LIN {X 0,Y 188.543,Z 754.958,A -85,B 0,C 180,E1 -22070.169,E2 -22070.169} C_VEL
LIN {X 0,Y 190.971,Z 747.164,A -85,B 0,C 180,E1 -22073.069,E2 -22073.069} C_VEL
LIN {X 0,Y 193.636,Z 737.842,A -85,B 0,C 180,E1 -22075.819,E2 -22075.819} C_VEL
LIN {X 0,Y 196.619,Z 727.143,A -85,B 0,C 180,E1 -22078.268,E2 -22078.268} C_VEL
LIN {X 0,Y 199.32,Z 716.514,A -85,B 0,C 180,E1 -22080.162,E2 -22080.162} C_VEL
LIN {X 0,Y 201.799,Z 704.647,A -85,B 0,C 180,E1 -22081.786,E2 -22081.786} C_VEL
LIN {X 0,Y 203.932,Z 692.297,A -85,B 0,C 180,E1 -22083.02,E2 -22083.02} C_VEL
LIN {X 0,Y 205.572,Z 679.263,A -85,B 0,C 180,E1 -22083.923,E2 -22083.923} C_VEL
LIN {X 0,Y 206.507,Z 665.005,A -85,B 0,C 180,E1 -22084.513,E2 -22084.513} C_VEL
LIN {X 0,Y 208.41,Z 623.369,A -85,B 0,C 180,E1 -22085.857,E2 -22085.857} C_VEL
LIN {X 0,Y 206.584,Z 608.008,A -85,B 0,C 180,E1 -22086.831,E2 -22086.831} C_VEL
LIN {X 0,Y 200.505,Z 592.715,A -85,B 0,C 180,E1 -22088.711,E2 -22088.711} C_VEL
LIN {X 0,Y 194.742,Z 580.478,A -85,B 0,C 180,E1 -22090.545,E2 -22090.545} C_VEL
LIN {X 0,Y 188.91,Z 569.734,A -85,B 0,C 180,E1 -22092.487,E2 -22092.487} C_VEL
LIN {X 0,Y 186.505,Z 565.259,A -85,B 0,C 180,E1 -22093.393,E2 -22093.393} C_VEL
LIN {X 0,Y 185.509,Z 561.374,A -85,B 0,C 180,E1 -22096.038,E2 -22096.038} C_VEL
LIN {X 0,Y 185.527,Z 561.37,A -85,B 0,C 180,E1 -22099.911,E2 -22099.911} C_VEL
LIN {X 0,Y 185.557,Z 561.366,A -85,B 0,C 180,E1 -22102.699,E2 -22102.699} C_VEL
LIN {X 0,Y 185.542,Z 561.366,A -85,B 0,C 180,E1 -22107.975,E2 -22107.975} C_VEL
LIN {X 0,Y 185.579,Z 561.365,A -85,B 0,C 180,E1 -22110.575,E2 -22110.575} C_VEL
LIN {X 0,Y 185.577,Z 561.365,A -85,B 0,C 180,E1 -22115.381,E2 -22115.381} C_VEL
LIN {X 0,Y 185.67,Z 561.351,A -85,B 0,C 180,E1 -22121.134,E2 -22121.134} C_VEL
LIN {X 0,Y 185.689,Z 561.353,A -85,B 0,C 180,E1 -22124.637,E2 -22124.637} C_VEL
LIN {X 0,Y 185.92,Z 561.313,A -85,B 0,C 180,E1 -22129.359,E2 -22129.359} C_VEL
LIN {X 0,Y 185.956,Z 561.316,A -85,B 0,C 180,E1 -22133.49,E2 -22133.49} C_VEL
LIN {X 0,Y 186.203,Z 561.289,A -85,B 0,C 180,E1 -22137.837,E2 -22137.837} C_VEL
LIN {X 0,Y 186.402,Z 561.263,A -85,B 0,C 180,E1 -22140,E2 -22140} C_VEL
LIN {X 0,Y 185.918,Z 561.321,A -85,B 0,C 180,E1 -22144.336,E2 -22144.336} C_VEL
LIN {X 0,Y 185.983,Z 561.305,A -85,B 0,C 180,E1 -22148.694,E2 -22148.694} C_VEL
LIN {X 0,Y 185.725,Z 561.339,A -85,B 0,C 180,E1 -22153.124,E2 -22153.124} C_VEL
LIN {X 0,Y 185.687,Z 561.346,A -85,B 0,C 180,E1 -22157.626,E2 -22157.626} C_VEL
LIN {X 0,Y 185.594,Z 561.358,A -85,B 0,C 180,E1 -22162.252,E2 -22162.252} C_VEL
LIN {X 0,Y 185.56,Z 561.363,A -85,B 0,C 180,E1 -22167.033,E2 -22167.033} C_VEL
LIN {X 0,Y 185.577,Z 561.369,A -85,B 0,C 180,E1 -22169.494,E2 -22169.494} C_VEL
LIN {X 0,Y 185.517,Z 561.375,A -85,B 0,C 180,E1 -22174.629,E2 -22174.629} C_VEL
LIN {X 0,Y 185.542,Z 561.349,A -85,B 0,C 180,E1 -22177.305,E2 -22177.305} C_VEL
LIN {X 0,Y 185.502,Z 561.377,A -85,B 0,C 180,E1 -22180.737,E2 -22180.737} C_VEL
LIN {X 0,Y 185.557,Z 561.366,A -85,B 0,C 180,E1 -22186.024,E2 -22186.024} C_VEL
LIN {X 0,Y 185.54,Z 561.371,A -85,B 0,C 180,E1 -22190.642,E2 -22190.642} C_VEL
LIN {X 0,Y 186.562,Z 564.249,A -85,B 0,C 180,E1 -22191.08,E2 -22191.08} C_VEL
LIN {X 0,Y 188.397,Z 566.543,A -85,B 0,C 180,E1 -22191.68,E2 -22191.68} C_VEL
LIN {X 0,Y 190.496,Z 569.807,A -85,B 0,C 180,E1 -22192.378,E2 -22192.378} C_VEL
LIN {X 0,Y 198.121,Z 582.425,A -85,B 0,C 180,E1 -22194.771,E2 -22194.771} C_VEL
LIN {X 0,Y 202.401,Z 590.493,A -85,B 0,C 180,E1 -22196.048,E2 -22196.048} C_VEL
LIN {X 0,Y 208.127,Z 604.639,A -85,B 0,C 180,E1 -22197.782,E2 -22197.782} C_VEL
LIN {X 0,Y 209.093,Z 607.323,A -85,B 0,C 180,E1 -22198.074,E2 -22198.074} C_VEL
LIN {X 0,Y 206.377,Z 664.41,A -85,B 0,C 180,E1 -22199.96,E2 -22199.96} C_VEL
LIN {X 0,Y 205.136,Z 677.197,A -85,B 0,C 180,E1 -22200.724,E2 -22200.724} C_VEL
LIN {X 0,Y 203.324,Z 690.286,A -85,B 0,C 180,E1 -22201.905,E2 -22201.905} C_VEL
LIN {X 0,Y 201.181,Z 701.437,A -85,B 0,C 180,E1 -22203.272,E2 -22203.272} C_VEL
LIN {X 0,Y 198.677,Z 712.971,A -85,B 0,C 180,E1 -22205.162,E2 -22205.162} C_VEL
LIN {X 0,Y 195.999,Z 723.355,A -85,B 0,C 180,E1 -22207.328,E2 -22207.328} C_VEL
LIN {X 0,Y 193.122,Z 732.726,A -85,B 0,C 180,E1 -22209.775,E2 -22209.775} C_VEL
LIN {X 0,Y 190.815,Z 740.39,A -85,B 0,C 180,E1 -22212.311,E2 -22212.311} C_VEL
LIN {X 0,Y 188.536,Z 747.886,A -85,B 0,C 180,E1 -22215.427,E2 -22215.427} C_VEL
LIN {X 0,Y 186.376,Z 754.818,A -85,B 0,C 180,E1 -22219.132,E2 -22219.132} C_VEL
LIN {X 0,Y 184.945,Z 759.415,A -85,B 0,C 180,E1 -22222.357,E2 -22222.357} C_VEL
LIN {X 0,Y 183.877,Z 762.924,A -85,B 0,C 180,E1 -22225.616,E2 -22225.616} C_VEL
LIN {X 0,Y 183.516,Z 764.709,A -85,B 0,C 180,E1 -22227.805,E2 -22227.805} C_VEL
LIN {X 0,Y 183.255,Z 766.055,A -85,B 0,C 180,E1 -22230,E2 -22230} C_VEL
LIN {X 0,Y 183.11,Z 767.437,A -85,B 0,C 180,E1 -22233.693,E2 -22233.693} C_VEL
LIN {X 0,Y 183.13,Z 767.766,A -85,B 0,C 180,E1 -22236.611,E2 -22236.611} C_VEL
LIN {X 0,Y 183.352,Z 767.525,A -85,B 0,C 180,E1 -22238.819,E2 -22238.819} C_VEL
LIN {X 0,Y 184.192,Z 765.895,A -85,B 0,C 180,E1 -22243.234,E2 -22243.234} C_VEL
LIN {X 0,Y 184.974,Z 764.457,A -85,B 0,C 180,E1 -22245.424,E2 -22245.424} C_VEL
LIN {X 0,Y 186.494,Z 761.495,A -85,B 0,C 180,E1 -22248.682,E2 -22248.682} C_VEL
LIN {X 0,Y 188.5,Z 757.475,A -85,B 0,C 180,E1 -22251.89,E2 -22251.89} C_VEL
LIN {X 0,Y 191.491,Z 751.27,A -85,B 0,C 180,E1 -22255.546,E2 -22255.546} C_VEL
LIN {X 0,Y 194.671,Z 744.497,A -85,B 0,C 180,E1 -22258.577,E2 -22258.577} C_VEL
LIN {X 0,Y 197.952,Z 736.516,A -85,B 0,C 180,E1 -22261.402,E2 -22261.402} C_VEL
LIN {X 0,Y 201.518,Z 727.312,A -85,B 0,C 180,E1 -22263.917,E2 -22263.917} C_VEL
LIN {X 0,Y 205.23,Z 716.545,A -85,B 0,C 180,E1 -22266.207,E2 -22266.207} C_VEL
LIN {X 0,Y 208.465,Z 705.768,A -85,B 0,C 180,E1 -22267.97,E2 -22267.97} C_VEL
LIN {X 0,Y 211.28,Z 693.797,A -85,B 0,C 180,E1 -22269.48,E2 -22269.48} C_VEL
LIN {X 0,Y 213.469,Z 681.932,A -85,B 0,C 180,E1 -22270.592,E2 -22270.592} C_VEL
LIN {X 0,Y 215.19,Z 668.883,A -85,B 0,C 180,E1 -22271.441,E2 -22271.441} C_VEL
LIN {X 0,Y 216.329,Z 654.16,A -85,B 0,C 180,E1 -22271.984,E2 -22271.984} C_VEL
LIN {X 0,Y 218.267,Z 616.856,A -85,B 0,C 180,E1 -22273.137,E2 -22273.137} C_VEL
LIN {X 0,Y 211.842,Z 602.253,A -85,B 0,C 180,E1 -22275.338,E2 -22275.338} C_VEL
LIN {X 0,Y 205.839,Z 590.838,A -85,B 0,C 180,E1 -22277.494,E2 -22277.494} C_VEL
LIN {X 0,Y 198.415,Z 579.63,A -85,B 0,C 180,E1 -22280.318,E2 -22280.318} C_VEL
LIN {X 0,Y 195.38,Z 575.413,A -85,B 0,C 180,E1 -22281.565,E2 -22281.565} C_VEL
LIN {X 0,Y 192.87,Z 571.791,A -85,B 0,C 180,E1 -22282.658,E2 -22282.658} C_VEL
LIN {X 0,Y 190.08,Z 568.518,A -85,B 0,C 180,E1 -22283.894,E2 -22283.894} C_VEL
LIN {X 0,Y 188.928,Z 566.576,A -85,B 0,C 180,E1 -22284.462,E2 -22284.462} C_VEL
LIN {X 0,Y 186.637,Z 564.42,A -85,B 0,C 180,E1 -22285.527,E2 -22285.527} C_VEL
LIN {X 0,Y 185.64,Z 561.964,A -85,B 0,C 180,E1 -22286.106,E2 -22286.106} C_VEL
LIN {X 0,Y 185.54,Z 561.367,A -85,B 0,C 180,E1 -22286.32,E2 -22286.32} C_VEL
LIN {X 0,Y 185.58,Z 561.363,A -85,B 0,C 180,E1 -22290.575,E2 -22290.575} C_VEL
LIN {X 0,Y 185.585,Z 561.369,A -85,B 0,C 180,E1 -22295.382,E2 -22295.382} C_VEL
LIN {X 0,Y 185.672,Z 561.35,A -85,B 0,C 180,E1 -22301.133,E2 -22301.133} C_VEL
LIN {X 0,Y 185.715,Z 561.353,A -85,B 0,C 180,E1 -22304.639,E2 -22304.639} C_VEL
LIN {X 0,Y 185.885,Z 561.331,A -85,B 0,C 180,E1 -22309.417,E2 -22309.417} C_VEL
LIN {X 0,Y 185.944,Z 561.312,A -85,B 0,C 180,E1 -22313.489,E2 -22313.489} C_VEL
LIN {X 0,Y 186.203,Z 561.275,A -85,B 0,C 180,E1 -22317.837,E2 -22317.837} C_VEL
LIN {X 0,Y 186.405,Z 561.265,A -85,B 0,C 180,E1 -22320,E2 -22320} C_VEL
LIN {X 0,Y 185.915,Z 561.315,A -85,B 0,C 180,E1 -22324.336,E2 -22324.336} C_VEL
LIN {X 0,Y 185.979,Z 561.305,A -85,B 0,C 180,E1 -22328.694,E2 -22328.694} C_VEL
LIN {X 0,Y 185.726,Z 561.337,A -85,B 0,C 180,E1 -22333.123,E2 -22333.123} C_VEL
LIN {X 0,Y 185.686,Z 561.346,A -85,B 0,C 180,E1 -22337.625,E2 -22337.625} C_VEL
LIN {X 0,Y 185.577,Z 561.359,A -85,B 0,C 180,E1 -22342.254,E2 -22342.254} C_VEL
LIN {X 0,Y 185.557,Z 561.36,A -85,B 0,C 180,E1 -22347.033,E2 -22347.033} C_VEL
LIN {X 0,Y 185.576,Z 561.369,A -85,B 0,C 180,E1 -22349.493,E2 -22349.493} C_VEL
LIN {X 0,Y 185.533,Z 561.375,A -85,B 0,C 180,E1 -22354.955,E2 -22354.955} C_VEL
LIN {X 0,Y 185.546,Z 561.404,A -85,B 0,C 180,E1 -22355.284,E2 -22355.284} C_VEL
LIN {X 0,Y 186.553,Z 564.822,A -85,B 0,C 180,E1 -22358.109,E2 -22358.109} C_VEL
LIN {X 0,Y 189.029,Z 568.779,A -85,B 0,C 180,E1 -22359.358,E2 -22359.358} C_VEL
LIN {X 0,Y 190.838,Z 571.151,A -85,B 0,C 180,E1 -22360.197,E2 -22360.197} C_VEL
LIN {X 0,Y 194.628,Z 577.119,A -85,B 0,C 180,E1 -22361.915,E2 -22361.915} C_VEL
LIN {X 0,Y 198.66,Z 583.78,A -85,B 0,C 180,E1 -22363.627,E2 -22363.627} C_VEL
LIN {X 0,Y 203.815,Z 592.834,A -85,B 0,C 180,E1 -22365.668,E2 -22365.668} C_VEL
LIN {X 0,Y 209.17,Z 603.347,A -85,B 0,C 180,E1 -22367.662,E2 -22367.662} C_VEL
LIN {X 0,Y 215.585,Z 617.992,A -85,B 0,C 180,E1 -22369.932,E2 -22369.932} C_VEL
LIN {X 0,Y 217.171,Z 622.529,A -85,B 0,C 180,E1 -22370.5,E2 -22370.5} C_VEL
LIN {X 0,Y 217.782,Z 628.099,A -85,B 0,C 180,E1 -22370.878,E2 -22370.878} C_VEL
LIN {X 0,Y 217.131,Z 640.755,A -85,B 0,C 180,E1 -22371.271,E2 -22371.271} C_VEL
LIN {X 0,Y 216.313,Z 646.602,A -85,B 0,C 180,E1 -22371.332,E2 -22371.332} C_VEL
LIN {X 0,Y 210.84,Z 665.607,A -85,B 0,C 180,E1 -22370.897,E2 -22370.897} C_VEL
LIN {X 0,Y 209.934,Z 671.439,A -85,B 0,C 180,E1 -22370.98,E2 -22370.98} C_VEL
LIN {X 0,Y 208.52,Z 684.399,A -85,B 0,C 180,E1 -22371.623,E2 -22371.623} C_VEL
LIN {X 0,Y 206.245,Z 697.423,A -85,B 0,C 180,E1 -22372.63,E2 -22372.63} C_VEL
LIN {X 0,Y 203.129,Z 710.093,A -85,B 0,C 180,E1 -22373.973,E2 -22373.973} C_VEL
LIN {X 0,Y 199.691,Z 721.918,A -85,B 0,C 180,E1 -22375.73,E2 -22375.73} C_VEL
LIN {X 0,Y 196.016,Z 732.495,A -85,B 0,C 180,E1 -22377.77,E2 -22377.77} C_VEL
LIN {X 0,Y 192.616,Z 741.146,A -85,B 0,C 180,E1 -22379.888,E2 -22379.888} C_VEL
LIN {X 0,Y 189.192,Z 749.123,A -85,B 0,C 180,E1 -22382.333,E2 -22382.333} C_VEL
LIN {X 0,Y 185.687,Z 756.958,A -85,B 0,C 180,E1 -22385.397,E2 -22385.397} C_VEL
LIN {X 0,Y 182.715,Z 763.231,A -85,B 0,C 180,E1 -22388.568,E2 -22388.568} C_VEL
LIN {X 0,Y 180.205,Z 768.235,A -85,B 0,C 180,E1 -22391.821,E2 -22391.821} C_VEL
LIN {X 0,Y 178.325,Z 772.12,A -85,B 0,C 180,E1 -22395.157,E2 -22395.157} C_VEL
LIN {X 0,Y 177.06,Z 774.991,A -85,B 0,C 180,E1 -22398.553,E2 -22398.553} C_VEL
LIN {X 0,Y 176.141,Z 777.331,A -85,B 0,C 180,E1 -22403.125,E2 -22403.125} C_VEL
LIN {X 0,Y 175.947,Z 778.069,A -85,B 0,C 180,E1 -22406.963,E2 -22406.963} C_VEL
LIN {X 0,Y 176.093,Z 777.854,A -85,B 0,C 180,E1 -22410,E2 -22410} C_VEL
LIN {X 0,Y 175.995,Z 776.812,A -85,B 0,C 180,E1 -22413.319,E2 -22413.319} C_VEL
LIN {X 0,Y 176.139,Z 774.727,A -85,B 0,C 180,E1 -22416.875,E2 -22416.875} C_VEL
LIN {X 0,Y 176.682,Z 771.719,A -85,B 0,C 180,E1 -22420.311,E2 -22420.311} C_VEL
LIN {X 0,Y 177.657,Z 767.649,A -85,B 0,C 180,E1 -22423.73,E2 -22423.73} C_VEL
LIN {X 0,Y 179.592,Z 761.398,A -85,B 0,C 180,E1 -22427.654,E2 -22427.654} C_VEL
LIN {X 0,Y 181.882,Z 754.591,A -85,B 0,C 180,E1 -22430.941,E2 -22430.941} C_VEL
LIN {X 0,Y 184.41,Z 746.72,A -85,B 0,C 180,E1 -22433.956,E2 -22433.956} C_VEL
LIN {X 0,Y 187.232,Z 737.377,A -85,B 0,C 180,E1 -22436.771,E2 -22436.771} C_VEL
LIN {X 0,Y 190.398,Z 726.628,A -85,B 0,C 180,E1 -22439.28,E2 -22439.28} C_VEL
LIN {X 0,Y 193.188,Z 715.925,A -85,B 0,C 180,E1 -22441.224,E2 -22441.224} C_VEL
LIN {X 0,Y 195.789,Z 703.916,A -85,B 0,C 180,E1 -22442.882,E2 -22442.882} C_VEL
LIN {X 0,Y 197.999,Z 691.402,A -85,B 0,C 180,E1 -22444.143,E2 -22444.143} C_VEL
LIN {X 0,Y 199.612,Z 678.891,A -85,B 0,C 180,E1 -22445.013,E2 -22445.013} C_VEL
LIN {X 0,Y 200.571,Z 664.781,A -85,B 0,C 180,E1 -22445.607,E2 -22445.607} C_VEL
LIN {X 0,Y 202.495,Z 623.747,A -85,B 0,C 180,E1 -22446.968,E2 -22446.968} C_VEL
LIN {X 0,Y 200.95,Z 610.485,A -85,B 0,C 180,E1 -22447.846,E2 -22447.846} C_VEL
LIN {X 0,Y 194.42,Z 594.119,A -85,B 0,C 180,E1 -22449.992,E2 -22449.992} C_VEL
LIN {X 0,Y 189.073,Z 582.905,A -85,B 0,C 180,E1 -22451.805,E2 -22451.805} C_VEL
LIN {X 0,Y 183.9,Z 573.454,A -85,B 0,C 180,E1 -22453.637,E2 -22453.637} C_VEL
LIN {X 0,Y 181.303,Z 569.018,A -85,B 0,C 180,E1 -22454.602,E2 -22454.602} C_VEL
LIN {X 0,Y 179.143,Z 564.973,A -85,B 0,C 180,E1 -22455.517,E2 -22455.517} C_VEL
LIN {X 0,Y 178.451,Z 562.254,A -85,B 0,C 180,E1 -22457.59,E2 -22457.59} C_VEL
LIN {X 0,Y 178.485,Z 562.251,A -85,B 0,C 180,E1 -22461.952,E2 -22461.952} C_VEL
LIN {X 0,Y 178.489,Z 562.245,A -85,B 0,C 180,E1 -22466.547,E2 -22466.547} C_VEL
LIN {X 0,Y 178.52,Z 562.246,A -85,B 0,C 180,E1 -22470.006,E2 -22470.006} C_VEL
LIN {X 0,Y 178.517,Z 562.248,A -85,B 0,C 180,E1 -22474.886,E2 -22474.886} C_VEL
LIN {X 0,Y 178.618,Z 562.232,A -85,B 0,C 180,E1 -22480.785,E2 -22480.785} C_VEL
LIN {X 0,Y 178.656,Z 562.229,A -85,B 0,C 180,E1 -22486.348,E2 -22486.348} C_VEL
LIN {X 0,Y 178.955,Z 562.191,A -85,B 0,C 180,E1 -22490.962,E2 -22490.962} C_VEL
LIN {X 0,Y 179.149,Z 562.166,A -85,B 0,C 180,E1 -22497.752,E2 -22497.752} C_VEL
LIN {X 0,Y 179.365,Z 562.14,A -85,B 0,C 180,E1 -22500,E2 -22500} C_VEL
LIN {X 0,Y 178.865,Z 562.2,A -85,B 0,C 180,E1 -22504.508,E2 -22504.508} C_VEL
LIN {X 0,Y 178.91,Z 562.181,A -85,B 0,C 180,E1 -22509.041,E2 -22509.041} C_VEL
LIN {X 0,Y 178.653,Z 562.223,A -85,B 0,C 180,E1 -22513.653,E2 -22513.653} C_VEL
LIN {X 0,Y 178.62,Z 562.211,A -85,B 0,C 180,E1 -22519.217,E2 -22519.217} C_VEL
LIN {X 0,Y 178.532,Z 562.244,A -85,B 0,C 180,E1 -22525.125,E2 -22525.125} C_VEL
LIN {X 0,Y 178.477,Z 562.248,A -85,B 0,C 180,E1 -22530.792,E2 -22530.792} C_VEL
LIN {X 0,Y 178.494,Z 562.25,A -85,B 0,C 180,E1 -22534.226,E2 -22534.226} C_VEL
LIN {X 0,Y 178.425,Z 562.24,A -85,B 0,C 180,E1 -22539.067,E2 -22539.067} C_VEL
LIN {X 0,Y 178.432,Z 562.257,A -85,B 0,C 180,E1 -22542.036,E2 -22542.036} C_VEL
LIN {X 0,Y 178.484,Z 562.25,A -85,B 0,C 180,E1 -22545.136,E2 -22545.136} C_VEL
LIN {X 0,Y 178.499,Z 562.245,A -85,B 0,C 180,E1 -22548.643,E2 -22548.643} C_VEL
LIN {X 0,Y 179.449,Z 564.993,A -85,B 0,C 180,E1 -22549.095,E2 -22549.095} C_VEL
LIN {X 0,Y 181.523,Z 567.603,A -85,B 0,C 180,E1 -22549.845,E2 -22549.845} C_VEL
LIN {X 0,Y 189.101,Z 579.424,A -85,B 0,C 180,E1 -22552.491,E2 -22552.491} C_VEL
LIN {X 0,Y 195.983,Z 591.447,A -85,B 0,C 180,E1 -22554.699,E2 -22554.699} C_VEL
LIN {X 0,Y 200.329,Z 601.448,A -85,B 0,C 180,E1 -22556.09,E2 -22556.09} C_VEL
LIN {X 0,Y 203.222,Z 609.307,A -85,B 0,C 180,E1 -22557.021,E2 -22557.021} C_VEL
LIN {X 0,Y 200.4,Z 664.717,A -85,B 0,C 180,E1 -22558.884,E2 -22558.884} C_VEL
LIN {X 0,Y 199.102,Z 677.541,A -85,B 0,C 180,E1 -22559.669,E2 -22559.669} C_VEL
LIN {X 0,Y 197.301,Z 690.057,A -85,B 0,C 180,E1 -22560.821,E2 -22560.821} C_VEL
LIN {X 0,Y 194.893,Z 702.123,A -85,B 0,C 180,E1 -22562.337,E2 -22562.337} C_VEL
LIN {X 0,Y 192.28,Z 713.569,A -85,B 0,C 180,E1 -22564.276,E2 -22564.276} C_VEL
LIN {X 0,Y 189.504,Z 723.884,A -85,B 0,C 180,E1 -22566.505,E2 -22566.505} C_VEL
LIN {X 0,Y 186.493,Z 733.181,A -85,B 0,C 180,E1 -22569.023,E2 -22569.023} C_VEL
LIN {X 0,Y 184.087,Z 740.801,A -85,B 0,C 180,E1 -22571.642,E2 -22571.642} C_VEL
LIN {X 0,Y 181.685,Z 748.261,A -85,B 0,C 180,E1 -22574.865,E2 -22574.865} C_VEL
LIN {X 0,Y 179.978,Z 753.364,A -85,B 0,C 180,E1 -22577.597,E2 -22577.597} C_VEL
LIN {X 0,Y 178.331,Z 758.315,A -85,B 0,C 180,E1 -22580.93,E2 -22580.93} C_VEL
LIN {X 0,Y 177.182,Z 762.148,A -85,B 0,C 180,E1 -22584.309,E2 -22584.309} C_VEL
LIN {X 0,Y 176.425,Z 764.969,A -85,B 0,C 180,E1 -22587.717,E2 -22587.717} C_VEL
LIN {X 0,Y 176.159,Z 766.303,A -85,B 0,C 180,E1 -22590,E2 -22590} C_VEL
LIN {X 0,Y 176.017,Z 767.573,A -85,B 0,C 180,E1 -22593.432,E2 -22593.432} C_VEL
LIN {X 0,Y 176.07,Z 767.965,A -85,B 0,C 180,E1 -22596.877,E2 -22596.877} C_VEL
LIN {X 0,Y 176.294,Z 767.712,A -85,B 0,C 180,E1 -22599.175,E2 -22599.175} C_VEL
LIN {X 0,Y 177.23,Z 766.058,A -85,B 0,C 180,E1 -22603.764,E2 -22603.764} C_VEL
LIN {X 0,Y 178.084,Z 764.595,A -85,B 0,C 180,E1 -22606.036,E2 -22606.036} C_VEL
LIN {X 0,Y 179.726,Z 761.606,A -85,B 0,C 180,E1 -22609.413,E2 -22609.413} C_VEL
LIN {X 0,Y 181.861,Z 757.557,A -85,B 0,C 180,E1 -22612.733,E2 -22612.733} C_VEL
LIN {X 0,Y 185.044,Z 751.32,A -85,B 0,C 180,E1 -22616.504,E2 -22616.504} C_VEL
LIN {X 0,Y 188.434,Z 744.513,A -85,B 0,C 180,E1 -22619.615,E2 -22619.615} C_VEL
LIN {X 0,Y 191.614,Z 737.093,A -85,B 0,C 180,E1 -22622.319,E2 -22622.319} C_VEL
LIN {X 0,Y 194.879,Z 729.146,A -85,B 0,C 180,E1 -22624.61,E2 -22624.61} C_VEL
LIN {X 0,Y 198.697,Z 718.745,A -85,B 0,C 180,E1 -22626.962,E2 -22626.962} C_VEL
LIN {X 0,Y 201.998,Z 708.425,A -85,B 0,C 180,E1 -22628.774,E2 -22628.774} C_VEL
LIN {X 0,Y 204.996,Z 697.107,A -85,B 0,C 180,E1 -22630.322,E2 -22630.322} C_VEL
LIN {X 0,Y 207.435,Z 685.236,A -85,B 0,C 180,E1 -22631.55,E2 -22631.55} C_VEL
LIN {X 0,Y 209.407,Z 672.259,A -85,B 0,C 180,E1 -22632.479,E2 -22632.479} C_VEL
LIN {X 0,Y 210.657,Z 659.075,A -85,B 0,C 180,E1 -22633.069,E2 -22633.069} C_VEL
LIN {X 0,Y 212.881,Z 619.185,A -85,B 0,C 180,E1 -22634.313,E2 -22634.313} C_VEL
LIN {X 0,Y 207.065,Z 605.808,A -85,B 0,C 180,E1 -22636.432,E2 -22636.432} C_VEL
LIN {X 0,Y 201.713,Z 595.497,A -85,B 0,C 180,E1 -22638.464,E2 -22638.464} C_VEL
LIN {X 0,Y 194.761,Z 584.818,A -85,B 0,C 180,E1 -22641.255,E2 -22641.255} C_VEL
LIN {X 0,Y 188.988,Z 576.793,A -85,B 0,C 180,E1 -22643.817,E2 -22643.817} C_VEL
LIN {X 0,Y 186.401,Z 573.24,A -85,B 0,C 180,E1 -22645.066,E2 -22645.066} C_VEL
LIN {X 0,Y 183.213,Z 569.464,A -85,B 0,C 180,E1 -22646.669,E2 -22646.669} C_VEL
LIN {X 0,Y 182.324,Z 567.709,A -85,B 0,C 180,E1 -22647.185,E2 -22647.185} C_VEL
LIN {X 0,Y 179.848,Z 565.62,A -85,B 0,C 180,E1 -22648.489,E2 -22648.489} C_VEL
LIN {X 0,Y 178.666,Z 563.187,A -85,B 0,C 180,E1 -22649.245,E2 -22649.245} C_VEL
LIN {X 0,Y 178.485,Z 562.244,A -85,B 0,C 180,E1 -22649.463,E2 -22649.463} C_VEL
LIN {X 0,Y 178.532,Z 562.242,A -85,B 0,C 180,E1 -22654.875,E2 -22654.875} C_VEL
LIN {X 0,Y 178.62,Z 562.231,A -85,B 0,C 180,E1 -22660.783,E2 -22660.783} C_VEL
LIN {X 0,Y 178.659,Z 562.227,A -85,B 0,C 180,E1 -22664.016,E2 -22664.016} C_VEL
LIN {X 0,Y 178.831,Z 562.207,A -85,B 0,C 180,E1 -22669.256,E2 -22669.256} C_VEL
LIN {X 0,Y 178.907,Z 562.186,A -85,B 0,C 180,E1 -22673.232,E2 -22673.232} C_VEL
LIN {X 0,Y 179.149,Z 562.154,A -85,B 0,C 180,E1 -22677.751,E2 -22677.751} C_VEL
LIN {X 0,Y 179.368,Z 562.141,A -85,B 0,C 180,E1 -22680,E2 -22680} C_VEL
LIN {X 0,Y 178.862,Z 562.195,A -85,B 0,C 180,E1 -22684.507,E2 -22684.507} C_VEL
LIN {X 0,Y 178.907,Z 562.186,A -85,B 0,C 180,E1 -22689.04,E2 -22689.04} C_VEL
LIN {X 0,Y 178.654,Z 562.217,A -85,B 0,C 180,E1 -22693.652,E2 -22693.652} C_VEL
LIN {X 0,Y 178.619,Z 562.225,A -85,B 0,C 180,E1 -22699.215,E2 -22699.215} C_VEL
LIN {X 0,Y 178.517,Z 562.249,A -85,B 0,C 180,E1 -22705.114,E2 -22705.114} C_VEL
LIN {X 0,Y 178.52,Z 562.246,A -85,B 0,C 180,E1 -22709.994,E2 -22709.994} C_VEL
LIN {X 0,Y 178.481,Z 562.291,A -85,B 0,C 180,E1 -22712.781,E2 -22712.781} C_VEL
LIN {X 0,Y 179.157,Z 564.483,A -85,B 0,C 180,E1 -22714.738,E2 -22714.738} C_VEL
LIN {X 0,Y 181.931,Z 568.738,A -85,B 0,C 180,E1 -22716.351,E2 -22716.351} C_VEL
LIN {X 0,Y 183.617,Z 570.874,A -85,B 0,C 180,E1 -22717.247,E2 -22717.247} C_VEL
LIN {X 0,Y 187.046,Z 575.824,A -85,B 0,C 180,E1 -22719.003,E2 -22719.003} C_VEL
LIN {X 0,Y 191.309,Z 582.727,A -85,B 0,C 180,E1 -22721.051,E2 -22721.051} C_VEL
LIN {X 0,Y 196.417,Z 591.278,A -85,B 0,C 180,E1 -22723.299,E2 -22723.299} C_VEL
LIN {X 0,Y 203.053,Z 603.976,A -85,B 0,C 180,E1 -22726,E2 -22726} C_VEL
LIN {X 0,Y 208.827,Z 616.827,A -85,B 0,C 180,E1 -22728.201,E2 -22728.201} C_VEL
LIN {X 0,Y 211.911,Z 624.661,A -85,B 0,C 180,E1 -22729.339,E2 -22729.339} C_VEL
LIN {X 0,Y 212.386,Z 629.434,A -85,B 0,C 180,E1 -22729.669,E2 -22729.669} C_VEL
LIN {X 0,Y 209.934,Z 671.439,A -85,B 0,C 180,E1 -22730.98,E2 -22730.98} C_VEL
LIN {X 0,Y 208.922,Z 677.25,A -85,B 0,C 180,E1 -22731.102,E2 -22731.102} C_VEL
LIN {X 0,Y 205.542,Z 686.583,A -85,B 0,C 180,E1 -22731.118,E2 -22731.118} C_VEL
LIN {X 0,Y 201.671,Z 695.687,A -85,B 0,C 180,E1 -22731.312,E2 -22731.312} C_VEL
LIN {X 0,Y 199.897,Z 701.137,A -85,B 0,C 180,E1 -22731.721,E2 -22731.721} C_VEL
LIN {X 0,Y 196.534,Z 713.517,A -85,B 0,C 180,E1 -22733.205,E2 -22733.205} C_VEL
LIN {X 0,Y 193.042,Z 724.632,A -85,B 0,C 180,E1 -22735.013,E2 -22735.013} C_VEL
LIN {X 0,Y 189.656,Z 733.639,A -85,B 0,C 180,E1 -22736.868,E2 -22736.868} C_VEL
LIN {X 0,Y 185.754,Z 742.892,A -85,B 0,C 180,E1 -22739.286,E2 -22739.286} C_VEL
LIN {X 0,Y 181.619,Z 751.883,A -85,B 0,C 180,E1 -22742.332,E2 -22742.332} C_VEL
LIN {X 0,Y 178.219,Z 759.138,A -85,B 0,C 180,E1 -22745.54,E2 -22745.54} C_VEL
LIN {X 0,Y 175.162,Z 764.959,A -85,B 0,C 180,E1 -22748.832,E2 -22748.832} C_VEL
LIN {X 0,Y 172.695,Z 769.551,A -85,B 0,C 180,E1 -22752.229,E2 -22752.229} C_VEL
LIN {X 0,Y 170.949,Z 773.059,A -85,B 0,C 180,E1 -22755.72,E2 -22755.72} C_VEL
LIN {X 0,Y 170.084,Z 774.834,A -85,B 0,C 180,E1 -22758.077,E2 -22758.077} C_VEL
LIN {X 0,Y 169.093,Z 777.153,A -85,B 0,C 180,E1 -22762.837,E2 -22762.837} C_VEL
LIN {X 0,Y 168.857,Z 777.896,A -85,B 0,C 180,E1 -22767.32,E2 -22767.32} C_VEL
LIN {X 0,Y 169.002,Z 777.634,A -85,B 0,C 180,E1 -22770,E2 -22770} C_VEL
LIN {X 0,Y 168.891,Z 776.804,A -85,B 0,C 180,E1 -22772.921,E2 -22772.921} C_VEL
LIN {X 0,Y 169.073,Z 774.463,A -85,B 0,C 180,E1 -22777.163,E2 -22777.163} C_VEL
LIN {X 0,Y 169.675,Z 771.432,A -85,B 0,C 180,E1 -22780.742,E2 -22780.742} C_VEL
LIN {X 0,Y 170.714,Z 767.337,A -85,B 0,C 180,E1 -22784.3,E2 -22784.3} C_VEL
LIN {X 0,Y 172.814,Z 761.059,A -85,B 0,C 180,E1 -22788.371,E2 -22788.371} C_VEL
LIN {X 0,Y 175.262,Z 754.224,A -85,B 0,C 180,E1 -22791.772,E2 -22791.772} C_VEL
LIN {X 0,Y 177.792,Z 746.664,A -85,B 0,C 180,E1 -22794.762,E2 -22794.762} C_VEL
LIN {X 0,Y 180.29,Z 738.829,A -85,B 0,C 180,E1 -22797.26,E2 -22797.26} C_VEL
LIN {X 0,Y 183.504,Z 728.471,A -85,B 0,C 180,E1 -22799.859,E2 -22799.859} C_VEL
LIN {X 0,Y 186.752,Z 716.78,A -85,B 0,C 180,E1 -22802.11,E2 -22802.11} C_VEL
LIN {X 0,Y 189.44,Z 705.179,A -85,B 0,C 180,E1 -22803.812,E2 -22803.812} C_VEL
LIN {X 0,Y 191.738,Z 693.121,A -85,B 0,C 180,E1 -22805.1,E2 -22805.1} C_VEL
LIN {X 0,Y 193.586,Z 679.798,A -85,B 0,C 180,E1 -22806.092,E2 -22806.092} C_VEL
LIN {X 0,Y 194.59,Z 666.927,A -85,B 0,C 180,E1 -22806.688,E2 -22806.688} C_VEL
LIN {X 0,Y 196.673,Z 624.509,A -85,B 0,C 180,E1 -22808.126,E2 -22808.126} C_VEL
LIN {X 0,Y 195.356,Z 612.972,A -85,B 0,C 180,E1 -22808.925,E2 -22808.925} C_VEL
LIN {X 0,Y 189.489,Z 598.045,A -85,B 0,C 180,E1 -22810.974,E2 -22810.974} C_VEL
LIN {X 0,Y 184.22,Z 586.787,A -85,B 0,C 180,E1 -22812.873,E2 -22812.873} C_VEL
LIN {X 0,Y 177.624,Z 574.578,A -85,B 0,C 180,E1 -22815.395,E2 -22815.395} C_VEL
LIN {X 0,Y 174.315,Z 569.191,A -85,B 0,C 180,E1 -22816.733,E2 -22816.733} C_VEL
LIN {X 0,Y 171.805,Z 564.712,A -85,B 0,C 180,E1 -22817.875,E2 -22817.875} C_VEL
LIN {X 0,Y 171.365,Z 563.134,A -85,B 0,C 180,E1 -22819.289,E2 -22819.289} C_VEL
LIN {X 0,Y 171.433,Z 563.129,A -85,B 0,C 180,E1 -22822.053,E2 -22822.053} C_VEL
LIN {X 0,Y 171.425,Z 563.123,A -85,B 0,C 180,E1 -22827.794,E2 -22827.794} C_VEL
LIN {X 0,Y 171.446,Z 563.124,A -85,B 0,C 180,E1 -22830.534,E2 -22830.534} C_VEL
LIN {X 0,Y 171.442,Z 563.122,A -85,B 0,C 180,E1 -22835.799,E2 -22835.799} C_VEL
LIN {X 0,Y 171.574,Z 563.108,A -85,B 0,C 180,E1 -22840.871,E2 -22840.871} C_VEL
LIN {X 0,Y 171.573,Z 563.113,A -85,B 0,C 180,E1 -22845.773,E2 -22845.773} C_VEL
LIN {X 0,Y 171.884,Z 563.071,A -85,B 0,C 180,E1 -22850.587,E2 -22850.587} C_VEL
LIN {X 0,Y 171.815,Z 563.067,A -85,B 0,C 180,E1 -22855.308,E2 -22855.308} C_VEL
LIN {X 0,Y 172.328,Z 563.016,A -85,B 0,C 180,E1 -22860,E2 -22860} C_VEL
LIN {X 0,Y 171.814,Z 563.079,A -85,B 0,C 180,E1 -22864.693,E2 -22864.693} C_VEL
LIN {X 0,Y 171.846,Z 563.056,A -85,B 0,C 180,E1 -22869.416,E2 -22869.416} C_VEL
LIN {X 0,Y 171.572,Z 563.11,A -85,B 0,C 180,E1 -22874.228,E2 -22874.228} C_VEL
LIN {X 0,Y 171.541,Z 563.091,A -85,B 0,C 180,E1 -22879.562,E2 -22879.562} C_VEL
LIN {X 0,Y 171.467,Z 563.121,A -85,B 0,C 180,E1 -22885.617,E2 -22885.617} C_VEL
LIN {X 0,Y 171.44,Z 563.125,A -85,B 0,C 180,E1 -22890.588,E2 -22890.588} C_VEL
LIN {X 0,Y 171.405,Z 563.128,A -85,B 0,C 180,E1 -22895.032,E2 -22895.032} C_VEL
LIN {X 0,Y 171.384,Z 563.114,A -85,B 0,C 180,E1 -22898.82,E2 -22898.82} C_VEL
LIN {X 0,Y 171.386,Z 563.137,A -85,B 0,C 180,E1 -22904.197,E2 -22904.197} C_VEL
LIN {X 0,Y 171.405,Z 563.192,A -85,B 0,C 180,E1 -22906.404,E2 -22906.404} C_VEL
LIN {X 0,Y 172.315,Z 565.839,A -85,B 0,C 180,E1 -22906.87,E2 -22906.87} C_VEL
LIN {X 0,Y 174.674,Z 568.619,A -85,B 0,C 180,E1 -22907.809,E2 -22907.809} C_VEL
LIN {X 0,Y 177.021,Z 572.099,A -85,B 0,C 180,E1 -22908.743,E2 -22908.743} C_VEL
LIN {X 0,Y 184.89,Z 584.458,A -85,B 0,C 180,E1 -22911.646,E2 -22911.646} C_VEL
LIN {X 0,Y 191.442,Z 596.213,A -85,B 0,C 180,E1 -22913.867,E2 -22913.867} C_VEL
LIN {X 0,Y 196.1,Z 607.512,A -85,B 0,C 180,E1 -22915.45,E2 -22915.45} C_VEL
LIN {X 0,Y 197.379,Z 611.075,A -85,B 0,C 180,E1 -22915.887,E2 -22915.887} C_VEL
LIN {X 0,Y 194.504,Z 665.067,A -85,B 0,C 180,E1 -22917.746,E2 -22917.746} C_VEL
LIN {X 0,Y 193.138,Z 677.892,A -85,B 0,C 180,E1 -22918.55,E2 -22918.55} C_VEL
LIN {X 0,Y 191.161,Z 690.94,A -85,B 0,C 180,E1 -22919.788,E2 -22919.788} C_VEL
LIN {X 0,Y 188.668,Z 702.809,A -85,B 0,C 180,E1 -22921.341,E2 -22921.341} C_VEL
LIN {X 0,Y 185.933,Z 714.167,A -85,B 0,C 180,E1 -22923.33,E2 -22923.33} C_VEL
LIN {X 0,Y 183.054,Z 724.412,A -85,B 0,C 180,E1 -22925.625,E2 -22925.625} C_VEL
LIN {X 0,Y 179.908,Z 733.633,A -85,B 0,C 180,E1 -22928.216,E2 -22928.216} C_VEL
LIN {X 0,Y 177.395,Z 741.211,A -85,B 0,C 180,E1 -22930.923,E2 -22930.923} C_VEL
LIN {X 0,Y 174.857,Z 748.636,A -85,B 0,C 180,E1 -22934.259,E2 -22934.259} C_VEL
LIN {X 0,Y 172.483,Z 755.5,A -85,B 0,C 180,E1 -22938.245,E2 -22938.245} C_VEL
LIN {X 0,Y 170.908,Z 760.036,A -85,B 0,C 180,E1 -22941.725,E2 -22941.725} C_VEL
LIN {X 0,Y 169.735,Z 763.495,A -85,B 0,C 180,E1 -22945.25,E2 -22945.25} C_VEL
LIN {X 0,Y 169.336,Z 765.229,A -85,B 0,C 180,E1 -22947.621,E2 -22947.621} C_VEL
LIN {X 0,Y 169.065,Z 766.551,A -85,B 0,C 180,E1 -22950,E2 -22950} C_VEL
LIN {X 0,Y 168.931,Z 767.712,A -85,B 0,C 180,E1 -22953.16,E2 -22953.16} C_VEL
LIN {X 0,Y 168.986,Z 768.164,A -85,B 0,C 180,E1 -22957.167,E2 -22957.167} C_VEL
LIN {X 0,Y 169.256,Z 767.899,A -85,B 0,C 180,E1 -22959.56,E2 -22959.56} C_VEL
LIN {X 0,Y 170.285,Z 766.219,A -85,B 0,C 180,E1 -22964.337,E2 -22964.337} C_VEL
LIN {X 0,Y 171.207,Z 764.732,A -85,B 0,C 180,E1 -22966.699,E2 -22966.699} C_VEL
LIN {X 0,Y 172.993,Z 761.716,A -85,B 0,C 180,E1 -22970.201,E2 -22970.201} C_VEL
LIN {X 0,Y 175.261,Z 757.639,A -85,B 0,C 180,E1 -22973.64,E2 -22973.64} C_VEL
LIN {X 0,Y 178.639,Z 751.371,A -85,B 0,C 180,E1 -22977.533,E2 -22977.533} C_VEL
LIN {X 0,Y 182.26,Z 744.529,A -85,B 0,C 180,E1 -22980.725,E2 -22980.725} C_VEL
LIN {X 0,Y 186.003,Z 736.197,A -85,B 0,C 180,E1 -22983.771,E2 -22983.771} C_VEL
LIN {X 0,Y 189.824,Z 727.122,A -85,B 0,C 180,E1 -22986.325,E2 -22986.325} C_VEL
LIN {X 0,Y 193.473,Z 717.411,A -85,B 0,C 180,E1 -22988.467,E2 -22988.467} C_VEL
LIN {X 0,Y 196.979,Z 706.76,A -85,B 0,C 180,E1 -22990.291,E2 -22990.291} C_VEL
LIN {X 0,Y 200.03,Z 694.813,A -85,B 0,C 180,E1 -22991.878,E2 -22991.878} C_VEL
LIN {X 0,Y 202.486,Z 682.756,A -85,B 0,C 180,E1 -22993.048,E2 -22993.048} C_VEL
LIN {X 0,Y 204.379,Z 669.587,A -85,B 0,C 180,E1 -22993.942,E2 -22993.942} C_VEL
LIN {X 0,Y 205.627,Z 654.88,A -85,B 0,C 180,E1 -22994.502,E2 -22994.502} C_VEL
LIN {X 0,Y 207.565,Z 621.377,A -85,B 0,C 180,E1 -22995.563,E2 -22995.563} C_VEL
LIN {X 0,Y 202.16,Z 608.941,A -85,B 0,C 180,E1 -22997.657,E2 -22997.657} C_VEL
LIN {X 0,Y 197.481,Z 599.9,A -85,B 0,C 180,E1 -22999.542,E2 -22999.542} C_VEL
LIN {X 0,Y 191.111,Z 590.02,A -85,B 0,C 180,E1 -23002.244,E2 -23002.244} C_VEL
LIN {X 0,Y 185.628,Z 582.243,A -85,B 0,C 180,E1 -23004.816,E2 -23004.816} C_VEL
LIN {X 0,Y 182.679,Z 578.235,A -85,B 0,C 180,E1 -23006.322,E2 -23006.322} C_VEL
LIN {X 0,Y 179.996,Z 574.73,A -85,B 0,C 180,E1 -23007.777,E2 -23007.777} C_VEL
LIN {X 0,Y 179.248,Z 573.672,A -85,B 0,C 180,E1 -23008.206,E2 -23008.206} C_VEL
LIN {X 0,Y 176.798,Z 571.014,A -85,B 0,C 180,E1 -23009.613,E2 -23009.613} C_VEL
LIN {X 0,Y 175.598,Z 568.722,A -85,B 0,C 180,E1 -23010.414,E2 -23010.414} C_VEL
LIN {X 0,Y 173.027,Z 566.803,A -85,B 0,C 180,E1 -23011.988,E2 -23011.988} C_VEL
LIN {X 0,Y 171.757,Z 564.573,A -85,B 0,C 180,E1 -23012.921,E2 -23012.921} C_VEL
LIN {X 0,Y 171.436,Z 563.12,A -85,B 0,C 180,E1 -23013.285,E2 -23013.285} C_VEL
LIN {X 0,Y 171.459,Z 563.117,A -85,B 0,C 180,E1 -23018.351,E2 -23018.351} C_VEL
LIN {X 0,Y 171.576,Z 563.107,A -85,B 0,C 180,E1 -23020.871,E2 -23020.871} C_VEL
LIN {X 0,Y 171.587,Z 563.104,A -85,B 0,C 180,E1 -23025.773,E2 -23025.773} C_VEL
LIN {X 0,Y 171.844,Z 563.076,A -85,B 0,C 180,E1 -23030.584,E2 -23030.584} C_VEL
LIN {X 0,Y 171.813,Z 563.084,A -85,B 0,C 180,E1 -23035.307,E2 -23035.307} C_VEL
LIN {X 0,Y 172.33,Z 563.018,A -85,B 0,C 180,E1 -23040,E2 -23040} C_VEL
LIN {X 0,Y 171.811,Z 563.074,A -85,B 0,C 180,E1 -23044.692,E2 -23044.692} C_VEL
LIN {X 0,Y 171.844,Z 563.067,A -85,B 0,C 180,E1 -23049.415,E2 -23049.415} C_VEL
LIN {X 0,Y 171.572,Z 563.1,A -85,B 0,C 180,E1 -23054.227,E2 -23054.227} C_VEL
LIN {X 0,Y 171.538,Z 563.109,A -85,B 0,C 180,E1 -23059.559,E2 -23059.559} C_VEL
LIN {X 0,Y 171.456,Z 563.125,A -85,B 0,C 180,E1 -23065.609,E2 -23065.609} C_VEL
LIN {X 0,Y 171.494,Z 563.185,A -85,B 0,C 180,E1 -23069.911,E2 -23069.911} C_VEL
LIN {X 0,Y 171.59,Z 563.929,A -85,B 0,C 180,E1 -23070.569,E2 -23070.569} C_VEL
LIN {X 0,Y 172.758,Z 566.458,A -85,B 0,C 180,E1 -23071.473,E2 -23071.473} C_VEL
LIN {X 0,Y 176.652,Z 570.799,A -85,B 0,C 180,E1 -23073.941,E2 -23073.941} C_VEL
LIN {X 0,Y 179.585,Z 575.156,A -85,B 0,C 180,E1 -23075.704,E2 -23075.704} C_VEL
LIN {X 0,Y 181.117,Z 577.455,A -85,B 0,C 180,E1 -23076.574,E2 -23076.574} C_VEL
LIN {X 0,Y 184.772,Z 582.98,A -85,B 0,C 180,E1 -23078.524,E2 -23078.524} C_VEL
LIN {X 0,Y 188.24,Z 588.735,A -85,B 0,C 180,E1 -23080.259,E2 -23080.259} C_VEL
LIN {X 0,Y 193.089,Z 597.155,A -85,B 0,C 180,E1 -23082.503,E2 -23082.503} C_VEL
LIN {X 0,Y 198.732,Z 608.157,A -85,B 0,C 180,E1 -23084.925,E2 -23084.925} C_VEL
LIN {X 0,Y 204.034,Z 620.201,A -85,B 0,C 180,E1 -23087.074,E2 -23087.074} C_VEL
LIN {X 0,Y 206.878,Z 627.486,A -85,B 0,C 180,E1 -23088.189,E2 -23088.189} C_VEL
LIN {X 0,Y 207.054,Z 631.409,A -85,B 0,C 180,E1 -23088.418,E2 -23088.418} C_VEL
LIN {X 0,Y 204.381,Z 674.133,A -85,B 0,C 180,E1 -23089.8,E2 -23089.8} C_VEL
LIN {X 0,Y 202.611,Z 687.504,A -85,B 0,C 180,E1 -23090.553,E2 -23090.553} C_VEL
LIN {X 0,Y 200.158,Z 700.055,A -85,B 0,C 180,E1 -23091.608,E2 -23091.608} C_VEL
LIN {X 0,Y 199.897,Z 701.137,A -85,B 0,C 180,E1 -23091.721,E2 -23091.721} C_VEL
LIN {X 0,Y 198.002,Z 706.624,A -85,B 0,C 180,E1 -23092.204,E2 -23092.204} C_VEL
LIN {X 0,Y 193.33,Z 715.178,A -85,B 0,C 180,E1 -23092.815,E2 -23092.815} C_VEL
LIN {X 0,Y 188.386,Z 723.227,A -85,B 0,C 180,E1 -23093.619,E2 -23093.619} C_VEL
LIN {X 0,Y 186.088,Z 727.913,A -85,B 0,C 180,E1 -23094.398,E2 -23094.398} C_VEL
LIN {X 0,Y 182.063,Z 737.617,A -85,B 0,C 180,E1 -23096.628,E2 -23096.628} C_VEL
LIN {X 0,Y 178.155,Z 746.132,A -85,B 0,C 180,E1 -23099.148,E2 -23099.148} C_VEL
LIN {X 0,Y 174.042,Z 754.43,A -85,B 0,C 180,E1 -23102.33,E2 -23102.33} C_VEL
LIN {X 0,Y 170.639,Z 761.132,A -85,B 0,C 180,E1 -23105.679,E2 -23105.679} C_VEL
LIN {X 0,Y 167.631,Z 766.494,A -85,B 0,C 180,E1 -23109.123,E2 -23109.123} C_VEL
LIN {X 0,Y 165.172,Z 770.687,A -85,B 0,C 180,E1 -23112.672,E2 -23112.672} C_VEL
LIN {X 0,Y 164.025,Z 772.92,A -85,B 0,C 180,E1 -23115.103,E2 -23115.103} C_VEL
LIN {X 0,Y 163.128,Z 774.676,A -85,B 0,C 180,E1 -23117.561,E2 -23117.561} C_VEL
LIN {X 0,Y 162.022,Z 776.974,A -85,B 0,C 180,E1 -23122.523,E2 -23122.523} C_VEL
LIN {X 0,Y 161.792,Z 777.539,A -85,B 0,C 180,E1 -23125.016,E2 -23125.016} C_VEL
LIN {X 0,Y 161.77,Z 777.66,A -85,B 0,C 180,E1 -23127.738,E2 -23127.738} C_VEL
LIN {X 0,Y 161.911,Z 777.414,A -85,B 0,C 180,E1 -23130,E2 -23130} C_VEL
LIN {X 0,Y 161.812,Z 776.714,A -85,B 0,C 180,E1 -23132.615,E2 -23132.615} C_VEL
LIN {X 0,Y 161.848,Z 775.704,A -85,B 0,C 180,E1 -23134.982,E2 -23134.982} C_VEL
LIN {X 0,Y 161.999,Z 774.198,A -85,B 0,C 180,E1 -23137.478,E2 -23137.478} C_VEL
LIN {X 0,Y 162.673,Z 771.144,A -85,B 0,C 180,E1 -23141.21,E2 -23141.21} C_VEL
LIN {X 0,Y 163.794,Z 767.024,A -85,B 0,C 180,E1 -23144.918,E2 -23144.918} C_VEL
LIN {X 0,Y 166.075,Z 760.721,A -85,B 0,C 180,E1 -23149.145,E2 -23149.145} C_VEL
LIN {X 0,Y 168.68,Z 753.856,A -85,B 0,C 180,E1 -23152.668,E2 -23152.668} C_VEL
LIN {X 0,Y 171.2,Z 746.621,A -85,B 0,C 180,E1 -23155.627,E2 -23155.627} C_VEL
LIN {X 0,Y 173.988,Z 738.387,A -85,B 0,C 180,E1 -23158.334,E2 -23158.334} C_VEL
LIN {X 0,Y 177.355,Z 727.954,A -85,B 0,C 180,E1 -23161.006,E2 -23161.006} C_VEL
LIN {X 0,Y 180.754,Z 716.197,A -85,B 0,C 180,E1 -23163.311,E2 -23163.311} C_VEL
LIN {X 0,Y 183.587,Z 704.451,A -85,B 0,C 180,E1 -23165.044,E2 -23165.044} C_VEL
LIN {X 0,Y 185.955,Z 692.227,A -85,B 0,C 180,E1 -23166.362,E2 -23166.362} C_VEL
LIN {X 0,Y 187.867,Z 678.776,A -85,B 0,C 180,E1 -23167.36,E2 -23167.36} C_VEL
LIN {X 0,Y 188.924,Z 664.544,A -85,B 0,C 180,E1 -23167.992,E2 -23167.992} C_VEL
LIN {X 0,Y 190.957,Z 625.569,A -85,B 0,C 180,E1 -23169.335,E2 -23169.335} C_VEL
LIN {X 0,Y 189.81,Z 615.337,A -85,B 0,C 180,E1 -23170.078,E2 -23170.078} C_VEL
LIN {X 0,Y 183.907,Z 600.289,A -85,B 0,C 180,E1 -23172.278,E2 -23172.278} C_VEL
LIN {X 0,Y 178.638,Z 589.084,A -85,B 0,C 180,E1 -23174.313,E2 -23174.313} C_VEL
LIN {X 0,Y 173.234,Z 579.074,A -85,B 0,C 180,E1 -23176.522,E2 -23176.522} C_VEL
LIN {X 0,Y 169.85,Z 573.496,A -85,B 0,C 180,E1 -23177.982,E2 -23177.982} C_VEL
LIN {X 0,Y 167.485,Z 569.465,A -85,B 0,C 180,E1 -23179.069,E2 -23179.069} C_VEL
LIN {X 0,Y 164.971,Z 566.155,A -85,B 0,C 180,E1 -23180.223,E2 -23180.223} C_VEL
LIN {X 0,Y 164.443,Z 564.475,A -85,B 0,C 180,E1 -23180.553,E2 -23180.553} C_VEL
LIN {X 0,Y 164.375,Z 564.009,A -85,B 0,C 180,E1 -23181.112,E2 -23181.112} C_VEL
LIN {X 0,Y 164.333,Z 564.009,A -85,B 0,C 180,E1 -23186.223,E2 -23186.223} C_VEL
LIN {X 0,Y 164.403,Z 564.005,A -85,B 0,C 180,E1 -23189.137,E2 -23189.137} C_VEL
LIN {X 0,Y 164.403,Z 564.006,A -85,B 0,C 180,E1 -23194.692,E2 -23194.692} C_VEL
LIN {X 0,Y 164.481,Z 563.996,A -85,B 0,C 180,E1 -23200.051,E2 -23200.051} C_VEL
LIN {X 0,Y 164.52,Z 563.991,A -85,B 0,C 180,E1 -23205.149,E2 -23205.149} C_VEL
LIN {X 0,Y 164.798,Z 563.948,A -85,B 0,C 180,E1 -23210.178,E2 -23210.178} C_VEL
LIN {X 0,Y 164.846,Z 563.951,A -85,B 0,C 180,E1 -23212.652,E2 -23212.652} C_VEL
LIN {X 0,Y 165.045,Z 563.921,A -85,B 0,C 180,E1 -23217.56,E2 -23217.56} C_VEL
LIN {X 0,Y 165.291,Z 563.893,A -85,B 0,C 180,E1 -23220,E2 -23220} C_VEL
LIN {X 0,Y 164.763,Z 563.958,A -85,B 0,C 180,E1 -23224.894,E2 -23224.894} C_VEL
LIN {X 0,Y 164.83,Z 563.949,A -85,B 0,C 180,E1 -23227.349,E2 -23227.349} C_VEL
LIN {X 0,Y 164.7,Z 563.938,A -85,B 0,C 180,E1 -23231.062,E2 -23231.062} C_VEL
LIN {X 0,Y 164.48,Z 563.987,A -85,B 0,C 180,E1 -23237.404,E2 -23237.404} C_VEL
LIN {X 0,Y 164.471,Z 563.97,A -85,B 0,C 180,E1 -23239.99,E2 -23239.99} C_VEL
LIN {X 0,Y 164.391,Z 563.999,A -85,B 0,C 180,E1 -23246.135,E2 -23246.135} C_VEL
LIN {X 0,Y 164.374,Z 564.003,A -85,B 0,C 180,E1 -23251.229,E2 -23251.229} C_VEL
LIN {X 0,Y 164.313,Z 563.992,A -85,B 0,C 180,E1 -23256.785,E2 -23256.785} C_VEL
LIN {X 0,Y 164.305,Z 564.006,A -85,B 0,C 180,E1 -23259.913,E2 -23259.913} C_VEL
LIN {X 0,Y 164.333,Z 564.017,A -85,B 0,C 180,E1 -23263.848,E2 -23263.848} C_VEL
LIN {X 0,Y 165.222,Z 566.634,A -85,B 0,C 180,E1 -23264.362,E2 -23264.362} C_VEL
LIN {X 0,Y 167.112,Z 568.796,A -85,B 0,C 180,E1 -23265.21,E2 -23265.21} C_VEL
LIN {X 0,Y 167.79,Z 569.669,A -85,B 0,C 180,E1 -23265.512,E2 -23265.512} C_VEL
LIN {X 0,Y 169.975,Z 572.942,A -85,B 0,C 180,E1 -23266.486,E2 -23266.486} C_VEL
LIN {X 0,Y 171.328,Z 574.837,A -85,B 0,C 180,E1 -23267.061,E2 -23267.061} C_VEL
LIN {X 0,Y 176.599,Z 582.797,A -85,B 0,C 180,E1 -23269.199,E2 -23269.199} C_VEL
LIN {X 0,Y 182.36,Z 592.375,A -85,B 0,C 180,E1 -23271.365,E2 -23271.365} C_VEL
LIN {X 0,Y 187.334,Z 601.841,A -85,B 0,C 180,E1 -23273.134,E2 -23273.134} C_VEL
LIN {X 0,Y 191.621,Z 612.913,A -85,B 0,C 180,E1 -23274.688,E2 -23274.688} C_VEL
LIN {X 0,Y 188.7,Z 665.357,A -85,B 0,C 180,E1 -23276.535,E2 -23276.535} C_VEL
LIN {X 0,Y 187.259,Z 678.221,A -85,B 0,C 180,E1 -23277.358,E2 -23277.358} C_VEL
LIN {X 0,Y 185.296,Z 690.718,A -85,B 0,C 180,E1 -23278.567,E2 -23278.567} C_VEL
LIN {X 0,Y 182.863,Z 701.923,A -85,B 0,C 180,E1 -23280.025,E2 -23280.025} C_VEL
LIN {X 0,Y 180.05,Z 713.476,A -85,B 0,C 180,E1 -23282.07,E2 -23282.07} C_VEL
LIN {X 0,Y 176.995,Z 723.878,A -85,B 0,C 180,E1 -23284.418,E2 -23284.418} C_VEL
LIN {X 0,Y 173.999,Z 732.399,A -85,B 0,C 180,E1 -23286.809,E2 -23286.809} C_VEL
LIN {X 0,Y 171.197,Z 740.242,A -85,B 0,C 180,E1 -23289.578,E2 -23289.578} C_VEL
LIN {X 0,Y 168.49,Z 747.901,A -85,B 0,C 180,E1 -23293.024,E2 -23293.024} C_VEL
LIN {X 0,Y 166.202,Z 754.051,A -85,B 0,C 180,E1 -23296.553,E2 -23296.553} C_VEL
LIN {X 0,Y 164.351,Z 758.941,A -85,B 0,C 180,E1 -23300.151,E2 -23300.151} C_VEL
LIN {X 0,Y 163.099,Z 762.718,A -85,B 0,C 180,E1 -23303.816,E2 -23303.816} C_VEL
LIN {X 0,Y 162.25,Z 765.489,A -85,B 0,C 180,E1 -23307.517,E2 -23307.517} C_VEL
LIN {X 0,Y 161.973,Z 766.798,A -85,B 0,C 180,E1 -23310,E2 -23310} C_VEL
LIN {X 0,Y 161.852,Z 767.847,A -85,B 0,C 180,E1 -23312.895,E2 -23312.895} C_VEL
LIN {X 0,Y 161.92,Z 768.363,A -85,B 0,C 180,E1 -23317.482,E2 -23317.482} C_VEL
LIN {X 0,Y 162.205,Z 768.087,A -85,B 0,C 180,E1 -23319.98,E2 -23319.98} C_VEL
LIN {X 0,Y 163.357,Z 766.377,A -85,B 0,C 180,E1 -23324.959,E2 -23324.959} C_VEL
LIN {X 0,Y 164.36,Z 764.87,A -85,B 0,C 180,E1 -23327.416,E2 -23327.416} C_VEL
LIN {X 0,Y 166.267,Z 761.863,A -85,B 0,C 180,E1 -23331.018,E2 -23331.018} C_VEL
LIN {X 0,Y 168.729,Z 757.721,A -85,B 0,C 180,E1 -23334.615,E2 -23334.615} C_VEL
LIN {X 0,Y 172.317,Z 751.422,A -85,B 0,C 180,E1 -23338.634,E2 -23338.634} C_VEL
LIN {X 0,Y 176.155,Z 744.546,A -85,B 0,C 180,E1 -23341.912,E2 -23341.912} C_VEL
LIN {X 0,Y 179.826,Z 736.765,A -85,B 0,C 180,E1 -23344.842,E2 -23344.842} C_VEL
LIN {X 0,Y 184.112,Z 727.03,A -85,B 0,C 180,E1 -23347.643,E2 -23347.643} C_VEL
LIN {X 0,Y 187.935,Z 717.258,A -85,B 0,C 180,E1 -23349.821,E2 -23349.821} C_VEL
LIN {X 0,Y 191.603,Z 706.513,A -85,B 0,C 180,E1 -23351.668,E2 -23351.668} C_VEL
LIN {X 0,Y 194.761,Z 694.412,A -85,B 0,C 180,E1 -23353.283,E2 -23353.283} C_VEL
LIN {X 0,Y 197.323,Z 682.168,A -85,B 0,C 180,E1 -23354.465,E2 -23354.465} C_VEL
LIN {X 0,Y 199.163,Z 669.677,A -85,B 0,C 180,E1 -23355.307,E2 -23355.307} C_VEL
LIN {X 0,Y 200.472,Z 654.722,A -85,B 0,C 180,E1 -23355.878,E2 -23355.878} C_VEL
LIN {X 0,Y 202.322,Z 623.558,A -85,B 0,C 180,E1 -23356.887,E2 -23356.887} C_VEL
LIN {X 0,Y 197.597,Z 612.643,A -85,B 0,C 180,E1 -23358.837,E2 -23358.837} C_VEL
LIN {X 0,Y 193.475,Z 604.534,A -85,B 0,C 180,E1 -23360.602,E2 -23360.602} C_VEL
LIN {X 0,Y 187.291,Z 594.806,A -85,B 0,C 180,E1 -23363.385,E2 -23363.385} C_VEL
LIN {X 0,Y 182.319,Z 587.657,A -85,B 0,C 180,E1 -23365.857,E2 -23365.857} C_VEL
LIN {X 0,Y 179.448,Z 583.74,A -85,B 0,C 180,E1 -23367.407,E2 -23367.407} C_VEL
LIN {X 0,Y 176.455,Z 579.651,A -85,B 0,C 180,E1 -23369.148,E2 -23369.148} C_VEL
LIN {X 0,Y 173.847,Z 576.467,A -85,B 0,C 180,E1 -23370.757,E2 -23370.757} C_VEL
LIN {X 0,Y 173.02,Z 575.05,A -85,B 0,C 180,E1 -23371.326,E2 -23371.326} C_VEL
LIN {X 0,Y 170.279,Z 572.447,A -85,B 0,C 180,E1 -23373.148,E2 -23373.148} C_VEL
LIN {X 0,Y 168.725,Z 569.667,A -85,B 0,C 180,E1 -23374.375,E2 -23374.375} C_VEL
LIN {X 0,Y 166.155,Z 567.841,A -85,B 0,C 180,E1 -23376.307,E2 -23376.307} C_VEL
LIN {X 0,Y 164.821,Z 565.701,A -85,B 0,C 180,E1 -23377.515,E2 -23377.515} C_VEL
LIN {X 0,Y 164.396,Z 563.995,A -85,B 0,C 180,E1 -23378.033,E2 -23378.033} C_VEL
LIN {X 0,Y 164.5,Z 563.981,A -85,B 0,C 180,E1 -23382.598,E2 -23382.598} C_VEL
LIN {X 0,Y 164.7,Z 563.963,A -85,B 0,C 180,E1 -23388.939,E2 -23388.939} C_VEL
LIN {X 0,Y 164.827,Z 563.938,A -85,B 0,C 180,E1 -23392.65,E2 -23392.65} C_VEL
LIN {X 0,Y 165.044,Z 563.91,A -85,B 0,C 180,E1 -23397.559,E2 -23397.559} C_VEL
LIN {X 0,Y 165.293,Z 563.893,A -85,B 0,C 180,E1 -23400,E2 -23400} C_VEL
LIN {X 0,Y 164.76,Z 563.954,A -85,B 0,C 180,E1 -23404.894,E2 -23404.894} C_VEL
LIN {X 0,Y 164.827,Z 563.943,A -85,B 0,C 180,E1 -23407.349,E2 -23407.349} C_VEL
LIN {X 0,Y 164.699,Z 563.97,A -85,B 0,C 180,E1 -23411.061,E2 -23411.061} C_VEL
LIN {X 0,Y 164.479,Z 563.988,A -85,B 0,C 180,E1 -23417.403,E2 -23417.403} C_VEL
LIN {X 0,Y 164.47,Z 563.993,A -85,B 0,C 180,E1 -23419.989,E2 -23419.989} C_VEL
LIN {X 0,Y 164.434,Z 564.103,A -85,B 0,C 180,E1 -23425.662,E2 -23425.662} C_VEL
LIN {X 0,Y 165.13,Z 566.421,A -85,B 0,C 180,E1 -23426.439,E2 -23426.439} C_VEL
LIN {X 0,Y 166.891,Z 568.619,A -85,B 0,C 180,E1 -23427.936,E2 -23427.936} C_VEL
LIN {X 0,Y 169.032,Z 570.017,A -85,B 0,C 180,E1 -23429.501,E2 -23429.501} C_VEL
LIN {X 0,Y 170.666,Z 572.948,A -85,B 0,C 180,E1 -23430.775,E2 -23430.775} C_VEL
LIN {X 0,Y 173.959,Z 576.687,A -85,B 0,C 180,E1 -23432.966,E2 -23432.966} C_VEL
LIN {X 0,Y 176.985,Z 581.229,A -85,B 0,C 180,E1 -23434.878,E2 -23434.878} C_VEL
LIN {X 0,Y 181.938,Z 589.063,A -85,B 0,C 180,E1 -23437.716,E2 -23437.716} C_VEL
LIN {X 0,Y 185.129,Z 594.551,A -85,B 0,C 180,E1 -23439.397,E2 -23439.397} C_VEL
LIN {X 0,Y 190.574,Z 604.394,A -85,B 0,C 180,E1 -23442.034,E2 -23442.034} C_VEL
LIN {X 0,Y 195.991,Z 615.663,A -85,B 0,C 180,E1 -23444.465,E2 -23444.465} C_VEL
LIN {X 0,Y 201.828,Z 630.004,A -85,B 0,C 180,E1 -23446.936,E2 -23446.936} C_VEL
LIN {X 0,Y 201.69,Z 635.58,A -85,B 0,C 180,E1 -23447.171,E2 -23447.171} C_VEL
LIN {X 0,Y 199.206,Z 673.602,A -85,B 0,C 180,E1 -23448.416,E2 -23448.416} C_VEL
LIN {X 0,Y 197.383,Z 687.047,A -85,B 0,C 180,E1 -23449.175,E2 -23449.175} C_VEL
LIN {X 0,Y 194.924,Z 699.338,A -85,B 0,C 180,E1 -23450.211,E2 -23450.211} C_VEL
LIN {X 0,Y 191.867,Z 710.575,A -85,B 0,C 180,E1 -23451.487,E2 -23451.487} C_VEL
LIN {X 0,Y 188.13,Z 722.193,A -85,B 0,C 180,E1 -23453.295,E2 -23453.295} C_VEL
LIN {X 0,Y 186.088,Z 727.913,A -85,B 0,C 180,E1 -23454.398,E2 -23454.398} C_VEL
LIN {X 0,Y 183.688,Z 732.552,A -85,B 0,C 180,E1 -23455.262,E2 -23455.262} C_VEL
LIN {X 0,Y 178.158,Z 739.727,A -85,B 0,C 180,E1 -23456.556,E2 -23456.556} C_VEL
LIN {X 0,Y 172.543,Z 746.338,A -85,B 0,C 180,E1 -23458.117,E2 -23458.117} C_VEL
LIN {X 0,Y 170.061,Z 750.086,A -85,B 0,C 180,E1 -23459.392,E2 -23459.392} C_VEL
LIN {X 0,Y 165.978,Z 757.657,A -85,B 0,C 180,E1 -23462.773,E2 -23462.773} C_VEL
LIN {X 0,Y 163.024,Z 762.975,A -85,B 0,C 180,E1 -23465.824,E2 -23465.824} C_VEL
LIN {X 0,Y 160.061,Z 767.902,A -85,B 0,C 180,E1 -23469.436,E2 -23469.436} C_VEL
LIN {X 0,Y 157.711,Z 771.714,A -85,B 0,C 180,E1 -23473.163,E2 -23473.163} C_VEL
LIN {X 0,Y 156.175,Z 774.519,A -85,B 0,C 180,E1 -23476.997,E2 -23476.997} C_VEL
LIN {X 0,Y 154.968,Z 776.795,A -85,B 0,C 180,E1 -23482.181,E2 -23482.181} C_VEL
LIN {X 0,Y 154.713,Z 777.345,A -85,B 0,C 180,E1 -23484.788,E2 -23484.788} C_VEL
LIN {X 0,Y 154.7,Z 777.424,A -85,B 0,C 180,E1 -23488.112,E2 -23488.112} C_VEL
LIN {X 0,Y 154.81,Z 777.193,A -85,B 0,C 180,E1 -23490,E2 -23490} C_VEL
LIN {X 0,Y 154.736,Z 776.525,A -85,B 0,C 180,E1 -23492.603,E2 -23492.603} C_VEL
LIN {X 0,Y 154.751,Z 775.458,A -85,B 0,C 180,E1 -23495.211,E2 -23495.211} C_VEL
LIN {X 0,Y 154.949,Z 773.934,A -85,B 0,C 180,E1 -23497.82,E2 -23497.82} C_VEL
LIN {X 0,Y 155.667,Z 770.856,A -85,B 0,C 180,E1 -23501.722,E2 -23501.722} C_VEL
LIN {X 0,Y 156.901,Z 766.711,A -85,B 0,C 180,E1 -23505.59,E2 -23505.59} C_VEL
LIN {X 0,Y 159.369,Z 760.382,A -85,B 0,C 180,E1 -23509.984,E2 -23509.984} C_VEL
LIN {X 0,Y 162.136,Z 753.488,A -85,B 0,C 180,E1 -23513.637,E2 -23513.637} C_VEL
LIN {X 0,Y 165.212,Z 745.014,A -85,B 0,C 180,E1 -23517.144,E2 -23517.144} C_VEL
LIN {X 0,Y 168.409,Z 735.983,A -85,B 0,C 180,E1 -23520.051,E2 -23520.051} C_VEL
LIN {X 0,Y 172.052,Z 725.075,A -85,B 0,C 180,E1 -23522.767,E2 -23522.767} C_VEL
LIN {X 0,Y 175.237,Z 714.066,A -85,B 0,C 180,E1 -23524.854,E2 -23524.854} C_VEL
LIN {X 0,Y 178.249,Z 701.716,A -85,B 0,C 180,E1 -23526.608,E2 -23526.608} C_VEL
LIN {X 0,Y 180.498,Z 690.017,A -85,B 0,C 180,E1 -23527.824,E2 -23527.824} C_VEL
LIN {X 0,Y 182.26,Z 677.22,A -85,B 0,C 180,E1 -23528.734,E2 -23528.734} C_VEL
LIN {X 0,Y 183.447,Z 660.645,A -85,B 0,C 180,E1 -23529.427,E2 -23529.427} C_VEL
LIN {X 0,Y 185.282,Z 626.064,A -85,B 0,C 180,E1 -23530.657,E2 -23530.657} C_VEL
LIN {X 0,Y 184.49,Z 618.207,A -85,B 0,C 180,E1 -23531.238,E2 -23531.238} C_VEL
LIN {X 0,Y 179.134,Z 604.213,A -85,B 0,C 180,E1 -23533.374,E2 -23533.374} C_VEL
LIN {X 0,Y 173.557,Z 592.154,A -85,B 0,C 180,E1 -23535.681,E2 -23535.681} C_VEL
LIN {X 0,Y 168.444,Z 582.75,A -85,B 0,C 180,E1 -23537.919,E2 -23537.919} C_VEL
LIN {X 0,Y 163.626,Z 574.509,A -85,B 0,C 180,E1 -23540.21,E2 -23540.21} C_VEL
LIN {X 0,Y 161.262,Z 571.264,A -85,B 0,C 180,E1 -23541.369,E2 -23541.369} C_VEL
LIN {X 0,Y 160.405,Z 569.88,A -85,B 0,C 180,E1 -23541.819,E2 -23541.819} C_VEL
LIN {X 0,Y 158.293,Z 567.718,A -85,B 0,C 180,E1 -23542.88,E2 -23542.88} C_VEL
LIN {X 0,Y 157.374,Z 565.38,A -85,B 0,C 180,E1 -23543.458,E2 -23543.458} C_VEL
LIN {X 0,Y 157.307,Z 564.882,A -85,B 0,C 180,E1 -23543.53,E2 -23543.53} C_VEL
LIN {X 0,Y 157.3,Z 564.883,A -85,B 0,C 180,E1 -23548.09,E2 -23548.09} C_VEL
LIN {X 0,Y 157.312,Z 564.885,A -85,B 0,C 180,E1 -23553.464,E2 -23553.464} C_VEL
LIN {X 0,Y 157.39,Z 564.881,A -85,B 0,C 180,E1 -23559.669,E2 -23559.669} C_VEL
LIN {X 0,Y 157.449,Z 564.869,A -85,B 0,C 180,E1 -23564.466,E2 -23564.466} C_VEL
LIN {X 0,Y 157.722,Z 564.825,A -85,B 0,C 180,E1 -23569.733,E2 -23569.733} C_VEL
LIN {X 0,Y 157.804,Z 564.828,A -85,B 0,C 180,E1 -23572.322,E2 -23572.322} C_VEL
LIN {X 0,Y 158.253,Z 564.77,A -85,B 0,C 180,E1 -23580,E2 -23580} C_VEL
LIN {X 0,Y 157.767,Z 564.827,A -85,B 0,C 180,E1 -23587.68,E2 -23587.68} C_VEL
LIN {X 0,Y 157.634,Z 564.818,A -85,B 0,C 180,E1 -23591.237,E2 -23591.237} C_VEL
LIN {X 0,Y 157.45,Z 564.873,A -85,B 0,C 180,E1 -23595.535,E2 -23595.535} C_VEL
LIN {X 0,Y 157.368,Z 564.857,A -85,B 0,C 180,E1 -23600.934,E2 -23600.934} C_VEL
LIN {X 0,Y 157.312,Z 564.88,A -85,B 0,C 180,E1 -23606.685,E2 -23606.685} C_VEL
LIN {X 0,Y 157.277,Z 564.888,A -85,B 0,C 180,E1 -23612.428,E2 -23612.428} C_VEL
LIN {X 0,Y 157.282,Z 564.869,A -85,B 0,C 180,E1 -23616.458,E2 -23616.458} C_VEL
LIN {X 0,Y 157.211,Z 564.903,A -85,B 0,C 180,E1 -23620.891,E2 -23620.891} C_VEL
LIN {X 0,Y 158.109,Z 567.578,A -85,B 0,C 180,E1 -23621.486,E2 -23621.486} C_VEL
LIN {X 0,Y 160.074,Z 569.733,A -85,B 0,C 180,E1 -23622.488,E2 -23622.488} C_VEL
LIN {X 0,Y 160.878,Z 570.507,A -85,B 0,C 180,E1 -23622.878,E2 -23622.878} C_VEL
LIN {X 0,Y 162.967,Z 573.764,A -85,B 0,C 180,E1 -23623.941,E2 -23623.941} C_VEL
LIN {X 0,Y 164.435,Z 575.637,A -85,B 0,C 180,E1 -23624.632,E2 -23624.632} C_VEL
LIN {X 0,Y 169.67,Z 583.208,A -85,B 0,C 180,E1 -23626.989,E2 -23626.989} C_VEL
LIN {X 0,Y 176.354,Z 594.104,A -85,B 0,C 180,E1 -23629.741,E2 -23629.741} C_VEL
LIN {X 0,Y 182.157,Z 605.001,A -85,B 0,C 180,E1 -23631.953,E2 -23631.953} C_VEL
LIN {X 0,Y 185.965,Z 614.752,A -85,B 0,C 180,E1 -23633.42,E2 -23633.42} C_VEL
LIN {X 0,Y 182.97,Z 665.718,A -85,B 0,C 180,E1 -23635.251,E2 -23635.251} C_VEL
LIN {X 0,Y 181.478,Z 678.559,A -85,B 0,C 180,E1 -23636.095,E2 -23636.095} C_VEL
LIN {X 0,Y 179.309,Z 691.576,A -85,B 0,C 180,E1 -23637.39,E2 -23637.39} C_VEL
LIN {X 0,Y 176.418,Z 704.174,A -85,B 0,C 180,E1 -23639.143,E2 -23639.143} C_VEL
LIN {X 0,Y 173.416,Z 715.358,A -85,B 0,C 180,E1 -23641.233,E2 -23641.233} C_VEL
LIN {X 0,Y 170.26,Z 725.439,A -85,B 0,C 180,E1 -23643.658,E2 -23643.658} C_VEL
LIN {X 0,Y 166.852,Z 734.535,A -85,B 0,C 180,E1 -23646.413,E2 -23646.413} C_VEL
LIN {X 0,Y 164.072,Z 742.031,A -85,B 0,C 180,E1 -23649.306,E2 -23649.306} C_VEL
LIN {X 0,Y 161.272,Z 749.384,A -85,B 0,C 180,E1 -23652.894,E2 -23652.894} C_VEL
LIN {X 0,Y 158.647,Z 756.165,A -85,B 0,C 180,E1 -23657.203,E2 -23657.203} C_VEL
LIN {X 0,Y 156.879,Z 760.643,A -85,B 0,C 180,E1 -23660.979,E2 -23660.979} C_VEL
LIN {X 0,Y 155.611,Z 764.054,A -85,B 0,C 180,E1 -23664.818,E2 -23664.818} C_VEL
LIN {X 0,Y 155.167,Z 765.749,A -85,B 0,C 180,E1 -23667.404,E2 -23667.404} C_VEL
LIN {X 0,Y 154.883,Z 767.045,A -85,B 0,C 180,E1 -23670,E2 -23670} C_VEL
LIN {X 0,Y 154.777,Z 767.955,A -85,B 0,C 180,E1 -23672.602,E2 -23672.602} C_VEL
LIN {X 0,Y 154.744,Z 768.47,A -85,B 0,C 180,E1 -23675.211,E2 -23675.211} C_VEL
LIN {X 0,Y 155.176,Z 768.274,A -85,B 0,C 180,E1 -23680.437,E2 -23680.437} C_VEL
LIN {X 0,Y 155.704,Z 767.604,A -85,B 0,C 180,E1 -23683.043,E2 -23683.043} C_VEL
LIN {X 0,Y 156.449,Z 766.531,A -85,B 0,C 180,E1 -23685.636,E2 -23685.636} C_VEL
LIN {X 0,Y 157.548,Z 765.007,A -85,B 0,C 180,E1 -23688.195,E2 -23688.195} C_VEL
LIN {X 0,Y 160.172,Z 761.063,A -85,B 0,C 180,E1 -23692.862,E2 -23692.862} C_VEL
LIN {X 0,Y 163.266,Z 756.192,A -85,B 0,C 180,E1 -23696.871,E2 -23696.871} C_VEL
LIN {X 0,Y 167.338,Z 749.324,A -85,B 0,C 180,E1 -23700.962,E2 -23700.962} C_VEL
LIN {X 0,Y 171.468,Z 741.864,A -85,B 0,C 180,E1 -23704.302,E2 -23704.302} C_VEL
LIN {X 0,Y 175.193,Z 734.235,A -85,B 0,C 180,E1 -23706.993,E2 -23706.993} C_VEL
LIN {X 0,Y 179.372,Z 724.953,A -85,B 0,C 180,E1 -23709.545,E2 -23709.545} C_VEL
LIN {X 0,Y 183.432,Z 714.588,A -85,B 0,C 180,E1 -23711.735,E2 -23711.735} C_VEL
LIN {X 0,Y 187.285,Z 703.067,A -85,B 0,C 180,E1 -23713.592,E2 -23713.592} C_VEL
LIN {X 0,Y 190.222,Z 691.629,A -85,B 0,C 180,E1 -23715.027,E2 -23715.027} C_VEL
LIN {X 0,Y 192.768,Z 678.709,A -85,B 0,C 180,E1 -23716.174,E2 -23716.174} C_VEL
LIN {X 0,Y 194.56,Z 665.724,A -85,B 0,C 180,E1 -23716.925,E2 -23716.925} C_VEL
LIN {X 0,Y 197.18,Z 625.884,A -85,B 0,C 180,E1 -23718.277,E2 -23718.277} C_VEL
LIN {X 0,Y 193.168,Z 616.448,A -85,B 0,C 180,E1 -23720.051,E2 -23720.051} C_VEL
LIN {X 0,Y 189.57,Z 609.206,A -85,B 0,C 180,E1 -23721.693,E2 -23721.693} C_VEL
LIN {X 0,Y 182.8,Z 598.296,A -85,B 0,C 180,E1 -23724.963,E2 -23724.963} C_VEL
LIN {X 0,Y 176.826,Z 589.85,A -85,B 0,C 180,E1 -23728.222,E2 -23728.222} C_VEL
LIN {X 0,Y 173.511,Z 585.369,A -85,B 0,C 180,E1 -23730.246,E2 -23730.246} C_VEL
LIN {X 0,Y 170.862,Z 581.705,A -85,B 0,C 180,E1 -23732.019,E2 -23732.019} C_VEL
LIN {X 0,Y 167.655,Z 578.114,A -85,B 0,C 180,E1 -23734.309,E2 -23734.309} C_VEL
LIN {X 0,Y 166.572,Z 576.212,A -85,B 0,C 180,E1 -23735.21,E2 -23735.21} C_VEL
LIN {X 0,Y 163.809,Z 573.812,A -85,B 0,C 180,E1 -23737.452,E2 -23737.452} C_VEL
LIN {X 0,Y 162.223,Z 570.74,A -85,B 0,C 180,E1 -23739.058,E2 -23739.058} C_VEL
LIN {X 0,Y 159.43,Z 568.987,A -85,B 0,C 180,E1 -23741.801,E2 -23741.801} C_VEL
LIN {X 0,Y 157.867,Z 566.551,A -85,B 0,C 180,E1 -23743.761,E2 -23743.761} C_VEL
LIN {X 0,Y 157.465,Z 564.871,A -85,B 0,C 180,E1 -23744.55,E2 -23744.55} C_VEL
LIN {X 0,Y 157.687,Z 564.844,A -85,B 0,C 180,E1 -23749.73,E2 -23749.73} C_VEL
LIN {X 0,Y 157.764,Z 564.817,A -85,B 0,C 180,E1 -23752.32,E2 -23752.32} C_VEL
LIN {X 0,Y 158.255,Z 564.769,A -85,B 0,C 180,E1 -23760,E2 -23760} C_VEL
LIN {X 0,Y 157.764,Z 564.82,A -85,B 0,C 180,E1 -23767.68,E2 -23767.68} C_VEL
LIN {X 0,Y 157.634,Z 564.85,A -85,B 0,C 180,E1 -23771.236,E2 -23771.236} C_VEL
LIN {X 0,Y 157.449,Z 564.868,A -85,B 0,C 180,E1 -23775.534,E2 -23775.534} C_VEL
LIN {X 0,Y 157.444,Z 564.997,A -85,B 0,C 180,E1 -23779.175,E2 -23779.175} C_VEL
LIN {X 0,Y 158.208,Z 567.388,A -85,B 0,C 180,E1 -23780.374,E2 -23780.374} C_VEL
LIN {X 0,Y 159.967,Z 569.573,A -85,B 0,C 180,E1 -23782.437,E2 -23782.437} C_VEL
LIN {X 0,Y 162.338,Z 570.974,A -85,B 0,C 180,E1 -23784.709,E2 -23784.709} C_VEL
LIN {X 0,Y 163.787,Z 573.817,A -85,B 0,C 180,E1 -23786.176,E2 -23786.176} C_VEL
LIN {X 0,Y 166.278,Z 576.069,A -85,B 0,C 180,E1 -23788.22,E2 -23788.22} C_VEL
LIN {X 0,Y 166.903,Z 576.685,A -85,B 0,C 180,E1 -23788.705,E2 -23788.705} C_VEL
LIN {X 0,Y 168.966,Z 579.806,A -85,B 0,C 180,E1 -23790.322,E2 -23790.322} C_VEL
LIN {X 0,Y 171.438,Z 582.795,A -85,B 0,C 180,E1 -23792.048,E2 -23792.048} C_VEL
LIN {X 0,Y 175.312,Z 588.933,A -85,B 0,C 180,E1 -23794.606,E2 -23794.606} C_VEL
LIN {X 0,Y 178.992,Z 594.857,A -85,B 0,C 180,E1 -23796.794,E2 -23796.794} C_VEL
LIN {X 0,Y 184.557,Z 604.869,A -85,B 0,C 180,E1 -23799.809,E2 -23799.809} C_VEL
LIN {X 0,Y 190.407,Z 616.763,A -85,B 0,C 180,E1 -23802.677,E2 -23802.677} C_VEL
LIN {X 0,Y 195.275,Z 628.472,A -85,B 0,C 180,E1 -23804.916,E2 -23804.916} C_VEL
LIN {X 0,Y 196.834,Z 632.622,A -85,B 0,C 180,E1 -23805.611,E2 -23805.611} C_VEL
LIN {X 0,Y 194.089,Z 673.661,A -85,B 0,C 180,E1 -23806.987,E2 -23806.987} C_VEL
LIN {X 0,Y 192.164,Z 687.192,A -85,B 0,C 180,E1 -23807.762,E2 -23807.762} C_VEL
LIN {X 0,Y 189.547,Z 699.717,A -85,B 0,C 180,E1 -23808.844,E2 -23808.844} C_VEL
LIN {X 0,Y 186.386,Z 710.793,A -85,B 0,C 180,E1 -23810.134,E2 -23810.134} C_VEL
LIN {X 0,Y 182.49,Z 722.334,A -85,B 0,C 180,E1 -23811.963,E2 -23811.963} C_VEL
LIN {X 0,Y 178.375,Z 732.732,A -85,B 0,C 180,E1 -23814.122,E2 -23814.122} C_VEL
LIN {X 0,Y 174.538,Z 741.24,A -85,B 0,C 180,E1 -23816.382,E2 -23816.382} C_VEL
LIN {X 0,Y 170.061,Z 750.086,A -85,B 0,C 180,E1 -23819.392,E2 -23819.392} C_VEL
LIN {X 0,Y 167.604,Z 753.673,A -85,B 0,C 180,E1 -23820.77,E2 -23820.77} C_VEL
LIN {X 0,Y 162.037,Z 759.052,A -85,B 0,C 180,E1 -23822.949,E2 -23822.949} C_VEL
LIN {X 0,Y 156.607,Z 763.727,A -85,B 0,C 180,E1 -23825.409,E2 -23825.409} C_VEL
LIN {X 0,Y 154.431,Z 766.243,A -85,B 0,C 180,E1 -23827.195,E2 -23827.195} C_VEL
LIN {X 0,Y 151.648,Z 770.442,A -85,B 0,C 180,E1 -23831.071,E2 -23831.071} C_VEL
LIN {X 0,Y 150.253,Z 772.638,A -85,B 0,C 180,E1 -23833.702,E2 -23833.702} C_VEL
LIN {X 0,Y 149.221,Z 774.361,A -85,B 0,C 180,E1 -23836.38,E2 -23836.38} C_VEL
LIN {X 0,Y 147.916,Z 776.617,A -85,B 0,C 180,E1 -23841.805,E2 -23841.805} C_VEL
LIN {X 0,Y 147.636,Z 777.148,A -85,B 0,C 180,E1 -23844.537,E2 -23844.537} C_VEL
LIN {X 0,Y 147.63,Z 777.181,A -85,B 0,C 180,E1 -23848.637,E2 -23848.637} C_VEL
LIN {X 0,Y 147.643,Z 776.293,A -85,B 0,C 180,E1 -23852.728,E2 -23852.728} C_VEL
LIN {X 0,Y 147.683,Z 775.21,A -85,B 0,C 180,E1 -23855.461,E2 -23855.461} C_VEL
LIN {X 0,Y 147.897,Z 773.669,A -85,B 0,C 180,E1 -23858.196,E2 -23858.196} C_VEL
LIN {X 0,Y 148.678,Z 770.567,A -85,B 0,C 180,E1 -23862.281,E2 -23862.281} C_VEL
LIN {X 0,Y 150.037,Z 766.397,A -85,B 0,C 180,E1 -23866.323,E2 -23866.323} C_VEL
LIN {X 0,Y 152.691,Z 760.042,A -85,B 0,C 180,E1 -23870.898,E2 -23870.898} C_VEL
LIN {X 0,Y 155.59,Z 753.198,A -85,B 0,C 180,E1 -23874.65,E2 -23874.65} C_VEL
LIN {X 0,Y 158.886,Z 744.589,A -85,B 0,C 180,E1 -23878.319,E2 -23878.319} C_VEL
LIN {X 0,Y 162.271,Z 735.515,A -85,B 0,C 180,E1 -23881.313,E2 -23881.313} C_VEL
LIN {X 0,Y 165.709,Z 725.735,A -85,B 0,C 180,E1 -23883.824,E2 -23883.824} C_VEL
LIN {X 0,Y 169.026,Z 715.012,A -85,B 0,C 180,E1 -23885.965,E2 -23885.965} C_VEL
LIN {X 0,Y 172.135,Z 702.976,A -85,B 0,C 180,E1 -23887.764,E2 -23887.764} C_VEL
LIN {X 0,Y 174.688,Z 690.419,A -85,B 0,C 180,E1 -23889.133,E2 -23889.133} C_VEL
LIN {X 0,Y 176.539,Z 677.938,A -85,B 0,C 180,E1 -23890.063,E2 -23890.063} C_VEL
LIN {X 0,Y 177.767,Z 662.338,A -85,B 0,C 180,E1 -23890.75,E2 -23890.75} C_VEL
LIN {X 0,Y 179.742,Z 627.199,A -85,B 0,C 180,E1 -23892.02,E2 -23892.02} C_VEL
LIN {X 0,Y 179.11,Z 620.619,A -85,B 0,C 180,E1 -23892.528,E2 -23892.528} C_VEL
LIN {X 0,Y 173.552,Z 606.025,A -85,B 0,C 180,E1 -23894.911,E2 -23894.911} C_VEL
LIN {X 0,Y 168.406,Z 595.069,A -85,B 0,C 180,E1 -23897.199,E2 -23897.199} C_VEL
LIN {X 0,Y 164.229,Z 587.223,A -85,B 0,C 180,E1 -23899.17,E2 -23899.17} C_VEL
LIN {X 0,Y 160.036,Z 579.879,A -85,B 0,C 180,E1 -23901.299,E2 -23901.299} C_VEL
LIN {X 0,Y 157.494,Z 576.115,A -85,B 0,C 180,E1 -23902.643,E2 -23902.643} C_VEL
LIN {X 0,Y 154.77,Z 572.864,A -85,B 0,C 180,E1 -23904.122,E2 -23904.122} C_VEL
LIN {X 0,Y 153.743,Z 571.031,A -85,B 0,C 180,E1 -23904.752,E2 -23904.752} C_VEL
LIN {X 0,Y 151.45,Z 569.01,A -85,B 0,C 180,E1 -23906.061,E2 -23906.061} C_VEL
LIN {X 0,Y 150.325,Z 566.478,A -85,B 0,C 180,E1 -23906.858,E2 -23906.858} C_VEL
LIN {X 0,Y 150.211,Z 565.764,A -85,B 0,C 180,E1 -23907.048,E2 -23907.048} C_VEL
LIN {X 0,Y 150.239,Z 565.761,A -85,B 0,C 180,E1 -23912.72,E2 -23912.72} C_VEL
LIN {X 0,Y 150.347,Z 565.756,A -85,B 0,C 180,E1 -23919.209,E2 -23919.209} C_VEL
LIN {X 0,Y 150.356,Z 565.745,A -85,B 0,C 180,E1 -23923.713,E2 -23923.713} C_VEL
LIN {X 0,Y 150.645,Z 565.704,A -85,B 0,C 180,E1 -23929.245,E2 -23929.245} C_VEL
LIN {X 0,Y 150.738,Z 565.709,A -85,B 0,C 180,E1 -23931.96,E2 -23931.96} C_VEL
LIN {X 0,Y 151.214,Z 565.646,A -85,B 0,C 180,E1 -23940,E2 -23940} C_VEL
LIN {X 0,Y 150.704,Z 565.701,A -85,B 0,C 180,E1 -23948.043,E2 -23948.043} C_VEL
LIN {X 0,Y 150.575,Z 565.696,A -85,B 0,C 180,E1 -23951.438,E2 -23951.438} C_VEL
LIN {X 0,Y 150.359,Z 565.755,A -85,B 0,C 180,E1 -23956.287,E2 -23956.287} C_VEL
LIN {X 0,Y 150.349,Z 565.729,A -85,B 0,C 180,E1 -23960.793,E2 -23960.793} C_VEL
LIN {X 0,Y 150.243,Z 565.761,A -85,B 0,C 180,E1 -23967.283,E2 -23967.283} C_VEL
LIN {X 0,Y 150.217,Z 565.768,A -85,B 0,C 180,E1 -23972.635,E2 -23972.635} C_VEL
LIN {X 0,Y 150.193,Z 565.753,A -85,B 0,C 180,E1 -23977.468,E2 -23977.468} C_VEL
LIN {X 0,Y 150.976,Z 568.191,A -85,B 0,C 180,E1 -23978.083,E2 -23978.083} C_VEL
LIN {X 0,Y 152.842,Z 570.459,A -85,B 0,C 180,E1 -23979.217,E2 -23979.217} C_VEL
LIN {X 0,Y 153.96,Z 571.419,A -85,B 0,C 180,E1 -23979.839,E2 -23979.839} C_VEL
LIN {X 0,Y 155.984,Z 574.684,A -85,B 0,C 180,E1 -23981.033,E2 -23981.033} C_VEL
LIN {X 0,Y 157.721,Z 576.547,A -85,B 0,C 180,E1 -23981.944,E2 -23981.944} C_VEL
LIN {X 0,Y 160.2,Z 580.014,A -85,B 0,C 180,E1 -23983.236,E2 -23983.236} C_VEL
LIN {X 0,Y 166.144,Z 588.871,A -85,B 0,C 180,E1 -23986.093,E2 -23986.093} C_VEL
LIN {X 0,Y 172.845,Z 600.11,A -85,B 0,C 180,E1 -23988.999,E2 -23988.999} C_VEL
LIN {X 0,Y 177.996,Z 610.337,A -85,B 0,C 180,E1 -23991.084,E2 -23991.084} C_VEL
LIN {X 0,Y 180.348,Z 616.55,A -85,B 0,C 180,E1 -23992.055,E2 -23992.055} C_VEL
LIN {X 0,Y 177.671,Z 662.099,A -85,B 0,C 180,E1 -23993.699,E2 -23993.699} C_VEL
LIN {X 0,Y 176.31,Z 675.057,A -85,B 0,C 180,E1 -23994.435,E2 -23994.435} C_VEL
LIN {X 0,Y 174.302,Z 687.987,A -85,B 0,C 180,E1 -23995.634,E2 -23995.634} C_VEL
LIN {X 0,Y 171.621,Z 699.925,A -85,B 0,C 180,E1 -23997.14,E2 -23997.14} C_VEL
LIN {X 0,Y 168.848,Z 710.719,A -85,B 0,C 180,E1 -23998.998,E2 -23998.998} C_VEL
LIN {X 0,Y 165.829,Z 720.65,A -85,B 0,C 180,E1 -24001.179,E2 -24001.179} C_VEL
LIN {X 0,Y 162.506,Z 729.795,A -85,B 0,C 180,E1 -24003.687,E2 -24003.687} C_VEL
LIN {X 0,Y 159.113,Z 738.151,A -85,B 0,C 180,E1 -24006.577,E2 -24006.577} C_VEL
LIN {X 0,Y 155.96,Z 746.293,A -85,B 0,C 180,E1 -24010.247,E2 -24010.247} C_VEL
LIN {X 0,Y 153.196,Z 752.861,A -85,B 0,C 180,E1 -24014.023,E2 -24014.023} C_VEL
LIN {X 0,Y 151.079,Z 758.094,A -85,B 0,C 180,E1 -24017.917,E2 -24017.917} C_VEL
LIN {X 0,Y 149.322,Z 762.179,A -85,B 0,C 180,E1 -24021.883,E2 -24021.883} C_VEL
LIN {X 0,Y 148.556,Z 764.328,A -85,B 0,C 180,E1 -24024.571,E2 -24024.571} C_VEL
LIN {X 0,Y 148.087,Z 766.008,A -85,B 0,C 180,E1 -24027.28,E2 -24027.28} C_VEL
LIN {X 0,Y 147.678,Z 767.971,A -85,B 0,C 180,E1 -24031.982,E2 -24031.982} C_VEL
LIN {X 0,Y 147.65,Z 768.682,A -85,B 0,C 180,E1 -24035.463,E2 -24035.463} C_VEL
LIN {X 0,Y 148.171,Z 768.462,A -85,B 0,C 180,E1 -24040.937,E2 -24040.937} C_VEL
LIN {X 0,Y 148.742,Z 767.78,A -85,B 0,C 180,E1 -24043.665,E2 -24043.665} C_VEL
LIN {X 0,Y 149.572,Z 766.683,A -85,B 0,C 180,E1 -24046.375,E2 -24046.375} C_VEL
LIN {X 0,Y 150.774,Z 765.145,A -85,B 0,C 180,E1 -24049.043,E2 -24049.043} C_VEL
LIN {X 0,Y 153.383,Z 761.469,A -85,B 0,C 180,E1 -24053.594,E2 -24053.594} C_VEL
LIN {X 0,Y 156.898,Z 756.268,A -85,B 0,C 180,E1 -24058.055,E2 -24058.055} C_VEL
LIN {X 0,Y 161.249,Z 749.36,A -85,B 0,C 180,E1 -24062.269,E2 -24062.269} C_VEL
LIN {X 0,Y 165.586,Z 741.864,A -85,B 0,C 180,E1 -24065.703,E2 -24065.703} C_VEL
LIN {X 0,Y 169.538,Z 734.193,A -85,B 0,C 180,E1 -24068.447,E2 -24068.447} C_VEL
LIN {X 0,Y 173.908,Z 724.833,A -85,B 0,C 180,E1 -24071.047,E2 -24071.047} C_VEL
LIN {X 0,Y 178.177,Z 714.401,A -85,B 0,C 180,E1 -24073.261,E2 -24073.261} C_VEL
LIN {X 0,Y 182.169,Z 702.79,A -85,B 0,C 180,E1 -24075.144,E2 -24075.144} C_VEL
LIN {X 0,Y 185.166,Z 691.503,A -85,B 0,C 180,E1 -24076.555,E2 -24076.555} C_VEL
LIN {X 0,Y 187.824,Z 678.453,A -85,B 0,C 180,E1 -24077.708,E2 -24077.708} C_VEL
LIN {X 0,Y 189.644,Z 665.555,A -85,B 0,C 180,E1 -24078.449,E2 -24078.449} C_VEL
LIN {X 0,Y 192.222,Z 628.255,A -85,B 0,C 180,E1 -24079.719,E2 -24079.719} C_VEL
LIN {X 0,Y 187.414,Z 617.087,A -85,B 0,C 180,E1 -24082.015,E2 -24082.015} C_VEL
LIN {X 0,Y 181.749,Z 607.154,A -85,B 0,C 180,E1 -24084.834,E2 -24084.834} C_VEL
LIN {X 0,Y 175.823,Z 598.287,A -85,B 0,C 180,E1 -24088.103,E2 -24088.103} C_VEL
LIN {X 0,Y 171.039,Z 591.485,A -85,B 0,C 180,E1 -24091.12,E2 -24091.12} C_VEL
LIN {X 0,Y 167.935,Z 587.328,A -85,B 0,C 180,E1 -24093.31,E2 -24093.31} C_VEL
LIN {X 0,Y 165.144,Z 583.832,A -85,B 0,C 180,E1 -24095.474,E2 -24095.474} C_VEL
LIN {X 0,Y 164.307,Z 582.582,A -85,B 0,C 180,E1 -24096.191,E2 -24096.191} C_VEL
LIN {X 0,Y 161.463,Z 579.613,A -85,B 0,C 180,E1 -24098.704,E2 -24098.704} C_VEL
LIN {X 0,Y 160.15,Z 577.343,A -85,B 0,C 180,E1 -24100.095,E2 -24100.095} C_VEL
LIN {X 0,Y 157.48,Z 575.174,A -85,B 0,C 180,E1 -24102.97,E2 -24102.97} C_VEL
LIN {X 0,Y 155.943,Z 572.243,A -85,B 0,C 180,E1 -24105.148,E2 -24105.148} C_VEL
LIN {X 0,Y 155.633,Z 571.709,A -85,B 0,C 180,E1 -24105.619,E2 -24105.619} C_VEL
LIN {X 0,Y 152.694,Z 569.894,A -85,B 0,C 180,E1 -24110.395,E2 -24110.395} C_VEL
LIN {X 0,Y 150.951,Z 566.9,A -85,B 0,C 180,E1 -24115.493,E2 -24115.493} C_VEL
LIN {X 0,Y 150.82,Z 565.685,A -85,B 0,C 180,E1 -24116.66,E2 -24116.66} C_VEL
LIN {X 0,Y 151.215,Z 565.645,A -85,B 0,C 180,E1 -24120,E2 -24120} C_VEL
LIN {X 0,Y 150.698,Z 565.897,A -85,B 0,C 180,E1 -24126.695,E2 -24126.695} C_VEL
LIN {X 0,Y 152.556,Z 569.927,A -85,B 0,C 180,E1 -24132.999,E2 -24132.999} C_VEL
LIN {X 0,Y 155.434,Z 571.69,A -85,B 0,C 180,E1 -24137.77,E2 -24137.77} C_VEL
LIN {X 0,Y 155.88,Z 572.099,A -85,B 0,C 180,E1 -24138.397,E2 -24138.397} C_VEL
LIN {X 0,Y 157.238,Z 574.999,A -85,B 0,C 180,E1 -24140.393,E2 -24140.393} C_VEL
LIN {X 0,Y 159.886,Z 577.27,A -85,B 0,C 180,E1 -24143.304,E2 -24143.304} C_VEL
LIN {X 0,Y 160.564,Z 577.87,A -85,B 0,C 180,E1 -24143.978,E2 -24143.978} C_VEL
LIN {X 0,Y 162.566,Z 581.088,A -85,B 0,C 180,E1 -24145.989,E2 -24145.989} C_VEL
LIN {X 0,Y 164.815,Z 583.226,A -85,B 0,C 180,E1 -24147.881,E2 -24147.881} C_VEL
LIN {X 0,Y 167.352,Z 586.722,A -85,B 0,C 180,E1 -24149.913,E2 -24149.913} C_VEL
LIN {X 0,Y 169.041,Z 589.108,A -85,B 0,C 180,E1 -24151.167,E2 -24151.167} C_VEL
LIN {X 0,Y 172.561,Z 594.768,A -85,B 0,C 180,E1 -24153.617,E2 -24153.617} C_VEL
LIN {X 0,Y 176.017,Z 600.587,A -85,B 0,C 180,E1 -24155.8,E2 -24155.8} C_VEL
LIN {X 0,Y 181.456,Z 610.68,A -85,B 0,C 180,E1 -24158.916,E2 -24158.916} C_VEL
LIN {X 0,Y 187.047,Z 622.652,A -85,B 0,C 180,E1 -24161.822,E2 -24161.822} C_VEL
LIN {X 0,Y 191.775,Z 634.689,A -85,B 0,C 180,E1 -24164.13,E2 -24164.13} C_VEL
LIN {X 0,Y 189.651,Z 667.768,A -85,B 0,C 180,E1 -24165.245,E2 -24165.245} C_VEL
LIN {X 0,Y 188.086,Z 681.325,A -85,B 0,C 180,E1 -24165.876,E2 -24165.876} C_VEL
LIN {X 0,Y 185.756,Z 693.894,A -85,B 0,C 180,E1 -24166.8,E2 -24166.8} C_VEL
LIN {X 0,Y 182.615,Z 705.864,A -85,B 0,C 180,E1 -24168.036,E2 -24168.036} C_VEL
LIN {X 0,Y 178.972,Z 717.075,A -85,B 0,C 180,E1 -24169.615,E2 -24169.615} C_VEL
LIN {X 0,Y 174.594,Z 728.504,A -85,B 0,C 180,E1 -24171.766,E2 -24171.766} C_VEL
LIN {X 0,Y 170.398,Z 737.709,A -85,B 0,C 180,E1 -24174.004,E2 -24174.004} C_VEL
LIN {X 0,Y 165.31,Z 747.607,A -85,B 0,C 180,E1 -24177.177,E2 -24177.177} C_VEL
LIN {X 0,Y 160.889,Z 755.582,A -85,B 0,C 180,E1 -24180.567,E2 -24180.567} C_VEL
LIN {X 0,Y 157.756,Z 760.99,A -85,B 0,C 180,E1 -24183.545,E2 -24183.545} C_VEL
LIN {X 0,Y 154.431,Z 766.243,A -85,B 0,C 180,E1 -24187.195,E2 -24187.195} C_VEL
LIN {X 0,Y 152.367,Z 768.547,A -85,B 0,C 180,E1 -24189.073,E2 -24189.073} C_VEL
LIN {X 0,Y 147.514,Z 771.66,A -85,B 0,C 180,E1 -24192.155,E2 -24192.155} C_VEL
LIN {X 0,Y 143.039,Z 774.096,A -85,B 0,C 180,E1 -24195.522,E2 -24195.522} C_VEL
LIN {X 0,Y 141.63,Z 775.17,A -85,B 0,C 180,E1 -24197.786,E2 -24197.786} C_VEL
LIN {X 0,Y 140.866,Z 776.438,A -85,B 0,C 180,E1 -24201.392,E2 -24201.392} C_VEL
LIN {X 0,Y 140.557,Z 776.95,A -85,B 0,C 180,E1 -24204.261,E2 -24204.261} C_VEL
LIN {X 0,Y 140.569,Z 776.856,A -85,B 0,C 180,E1 -24209.356,E2 -24209.356} C_VEL
LIN {X 0,Y 140.547,Z 776.062,A -85,B 0,C 180,E1 -24212.866,E2 -24212.866} C_VEL
LIN {X 0,Y 140.614,Z 774.96,A -85,B 0,C 180,E1 -24215.737,E2 -24215.737} C_VEL
LIN {X 0,Y 140.847,Z 773.403,A -85,B 0,C 180,E1 -24218.609,E2 -24218.609} C_VEL
LIN {X 0,Y 141.716,Z 770.277,A -85,B 0,C 180,E1 -24222.895,E2 -24222.895} C_VEL
LIN {X 0,Y 143.199,Z 766.083,A -85,B 0,C 180,E1 -24227.125,E2 -24227.125} C_VEL
LIN {X 0,Y 146.044,Z 759.7,A -85,B 0,C 180,E1 -24231.897,E2 -24231.897} C_VEL
LIN {X 0,Y 149.325,Z 752.291,A -85,B 0,C 180,E1 -24236.064,E2 -24236.064} C_VEL
LIN {X 0,Y 152.672,Z 743.998,A -85,B 0,C 180,E1 -24239.66,E2 -24239.66} C_VEL
LIN {X 0,Y 156.234,Z 735.048,A -85,B 0,C 180,E1 -24242.669,E2 -24242.669} C_VEL
LIN {X 0,Y 159.824,Z 725.214,A -85,B 0,C 180,E1 -24245.249,E2 -24245.249} C_VEL
LIN {X 0,Y 163.295,Z 714.395,A -85,B 0,C 180,E1 -24247.438,E2 -24247.438} C_VEL
LIN {X 0,Y 166.552,Z 702.235,A -85,B 0,C 180,E1 -24249.267,E2 -24249.267} C_VEL
LIN {X 0,Y 169.21,Z 689.513,A -85,B 0,C 180,E1 -24250.659,E2 -24250.659} C_VEL
LIN {X 0,Y 171.128,Z 676.664,A -85,B 0,C 180,E1 -24251.592,E2 -24251.592} C_VEL
LIN {X 0,Y 172.463,Z 659.357,A -85,B 0,C 180,E1 -24252.333,E2 -24252.333} C_VEL
LIN {X 0,Y 174.326,Z 628.15,A -85,B 0,C 180,E1 -24253.475,E2 -24253.475} C_VEL
LIN {X 0,Y 173.799,Z 622.949,A -85,B 0,C 180,E1 -24253.91,E2 -24253.91} C_VEL
LIN {X 0,Y 168.82,Z 609.689,A -85,B 0,C 180,E1 -24256.203,E2 -24256.203} C_VEL
LIN {X 0,Y 163.689,Z 598.485,A -85,B 0,C 180,E1 -24258.665,E2 -24258.665} C_VEL
LIN {X 0,Y 158.685,Z 589.041,A -85,B 0,C 180,E1 -24261.241,E2 -24261.241} C_VEL
LIN {X 0,Y 156.186,Z 584.844,A -85,B 0,C 180,E1 -24262.607,E2 -24262.607} C_VEL
LIN {X 0,Y 153.425,Z 580.927,A -85,B 0,C 180,E1 -24264.164,E2 -24264.164} C_VEL
LIN {X 0,Y 150.517,Z 576.887,A -85,B 0,C 180,E1 -24265.923,E2 -24265.923} C_VEL
LIN {X 0,Y 148.202,Z 574.301,A -85,B 0,C 180,E1 -24267.378,E2 -24267.378} C_VEL
LIN {X 0,Y 146.972,Z 572.09,A -85,B 0,C 180,E1 -24268.264,E2 -24268.264} C_VEL
LIN {X 0,Y 144.441,Z 569.964,A -85,B 0,C 180,E1 -24269.984,E2 -24269.984} C_VEL
LIN {X 0,Y 143.38,Z 567.81,A -85,B 0,C 180,E1 -24270.867,E2 -24270.867} C_VEL
LIN {X 0,Y 143.14,Z 566.643,A -85,B 0,C 180,E1 -24271.251,E2 -24271.251} C_VEL
LIN {X 0,Y 143.177,Z 566.637,A -85,B 0,C 180,E1 -24276.878,E2 -24276.878} C_VEL
LIN {X 0,Y 143.303,Z 566.635,A -85,B 0,C 180,E1 -24279.922,E2 -24279.922} C_VEL
LIN {X 0,Y 143.36,Z 566.627,A -85,B 0,C 180,E1 -24285.812,E2 -24285.812} C_VEL
LIN {X 0,Y 143.592,Z 566.581,A -85,B 0,C 180,E1 -24288.71,E2 -24288.71} C_VEL
LIN {X 0,Y 143.658,Z 566.59,A -85,B 0,C 180,E1 -24291.561,E2 -24291.561} C_VEL
LIN {X 0,Y 144.173,Z 566.523,A -85,B 0,C 180,E1 -24300,E2 -24300} C_VEL
LIN {X 0,Y 143.624,Z 566.576,A -85,B 0,C 180,E1 -24308.442,E2 -24308.442} C_VEL
LIN {X 0,Y 143.502,Z 566.577,A -85,B 0,C 180,E1 -24311.629,E2 -24311.629} C_VEL
LIN {X 0,Y 143.293,Z 566.626,A -85,B 0,C 180,E1 -24317.115,E2 -24317.115} C_VEL
LIN {X 0,Y 143.275,Z 566.612,A -85,B 0,C 180,E1 -24321.255,E2 -24321.255} C_VEL
LIN {X 0,Y 143.189,Z 566.642,A -85,B 0,C 180,E1 -24327.938,E2 -24327.938} C_VEL
LIN {X 0,Y 143.171,Z 566.65,A -85,B 0,C 180,E1 -24333.279,E2 -24333.279} C_VEL
LIN {X 0,Y 144.079,Z 569.385,A -85,B 0,C 180,E1 -24334.19,E2 -24334.19} C_VEL
LIN {X 0,Y 145.967,Z 571.499,A -85,B 0,C 180,E1 -24335.548,E2 -24335.548} C_VEL
LIN {X 0,Y 147.26,Z 572.443,A -85,B 0,C 180,E1 -24336.389,E2 -24336.389} C_VEL
LIN {X 0,Y 149.066,Z 575.468,A -85,B 0,C 180,E1 -24337.649,E2 -24337.649} C_VEL
LIN {X 0,Y 150.983,Z 577.546,A -85,B 0,C 180,E1 -24338.826,E2 -24338.826} C_VEL
LIN {X 0,Y 153.689,Z 581.316,A -85,B 0,C 180,E1 -24340.448,E2 -24340.448} C_VEL
LIN {X 0,Y 158.033,Z 587.47,A -85,B 0,C 180,E1 -24342.835,E2 -24342.835} C_VEL
LIN {X 0,Y 162.996,Z 595.067,A -85,B 0,C 180,E1 -24345.319,E2 -24345.319} C_VEL
LIN {X 0,Y 168.761,Z 605.06,A -85,B 0,C 180,E1 -24347.965,E2 -24347.965} C_VEL
LIN {X 0,Y 173.415,Z 614.584,A -85,B 0,C 180,E1 -24349.976,E2 -24349.976} C_VEL
LIN {X 0,Y 174.93,Z 618.805,A -85,B 0,C 180,E1 -24350.655,E2 -24350.655} C_VEL
LIN {X 0,Y 171.918,Z 665.495,A -85,B 0,C 180,E1 -24352.379,E2 -24352.379} C_VEL
LIN {X 0,Y 170.284,Z 678.544,A -85,B 0,C 180,E1 -24353.25,E2 -24353.25} C_VEL
LIN {X 0,Y 168.037,Z 691.124,A -85,B 0,C 180,E1 -24354.529,E2 -24354.529} C_VEL
LIN {X 0,Y 165.294,Z 702.387,A -85,B 0,C 180,E1 -24356.08,E2 -24356.08} C_VEL
LIN {X 0,Y 162.035,Z 713.971,A -85,B 0,C 180,E1 -24358.272,E2 -24358.272} C_VEL
LIN {X 0,Y 158.51,Z 724.394,A -85,B 0,C 180,E1 -24360.81,E2 -24360.81} C_VEL
LIN {X 0,Y 154.714,Z 733.806,A -85,B 0,C 180,E1 -24363.712,E2 -24363.712} C_VEL
LIN {X 0,Y 151.5,Z 741.502,A -85,B 0,C 180,E1 -24366.778,E2 -24366.778} C_VEL
LIN {X 0,Y 148.302,Z 749.02,A -85,B 0,C 180,E1 -24370.627,E2 -24370.627} C_VEL
LIN {X 0,Y 145.629,Z 755.071,A -85,B 0,C 180,E1 -24374.608,E2 -24374.608} C_VEL
LIN {X 0,Y 143.471,Z 759.876,A -85,B 0,C 180,E1 -24378.701,E2 -24378.701} C_VEL
LIN {X 0,Y 141.967,Z 763.574,A -85,B 0,C 180,E1 -24382.891,E2 -24382.891} C_VEL
LIN {X 0,Y 141.009,Z 766.267,A -85,B 0,C 180,E1 -24387.143,E2 -24387.143} C_VEL
LIN {X 0,Y 140.605,Z 768.024,A -85,B 0,C 180,E1 -24391.431,E2 -24391.431} C_VEL
LIN {X 0,Y 140.557,Z 768.893,A -85,B 0,C 180,E1 -24395.739,E2 -24395.739} C_VEL
LIN {X 0,Y 140.745,Z 768.961,A -85,B 0,C 180,E1 -24398.615,E2 -24398.615} C_VEL
LIN {X 0,Y 141.808,Z 767.955,A -85,B 0,C 180,E1 -24404.347,E2 -24404.347} C_VEL
LIN {X 0,Y 142.73,Z 766.834,A -85,B 0,C 180,E1 -24407.183,E2 -24407.183} C_VEL
LIN {X 0,Y 144.022,Z 765.284,A -85,B 0,C 180,E1 -24409.973,E2 -24409.973} C_VEL
LIN {X 0,Y 146.591,Z 761.902,A -85,B 0,C 180,E1 -24414.366,E2 -24414.366} C_VEL
LIN {X 0,Y 149.453,Z 757.971,A -85,B 0,C 180,E1 -24418.05,E2 -24418.05} C_VEL
LIN {X 0,Y 153.802,Z 751.58,A -85,B 0,C 180,E1 -24422.473,E2 -24422.473} C_VEL
LIN {X 0,Y 158.29,Z 744.574,A -85,B 0,C 180,E1 -24426.035,E2 -24426.035} C_VEL
LIN {X 0,Y 162.431,Z 737.142,A -85,B 0,C 180,E1 -24428.988,E2 -24428.988} C_VEL
LIN {X 0,Y 166.711,Z 728.712,A -85,B 0,C 180,E1 -24431.602,E2 -24431.602} C_VEL
LIN {X 0,Y 171.515,Z 717.981,A -85,B 0,C 180,E1 -24434.153,E2 -24434.153} C_VEL
LIN {X 0,Y 175.649,Z 707.268,A -85,B 0,C 180,E1 -24436.07,E2 -24436.07} C_VEL
LIN {X 0,Y 179.247,Z 695.214,A -85,B 0,C 180,E1 -24437.735,E2 -24437.735} C_VEL
LIN {X 0,Y 182.17,Z 682.758,A -85,B 0,C 180,E1 -24438.974,E2 -24438.974} C_VEL
LIN {X 0,Y 184.238,Z 670.343,A -85,B 0,C 180,E1 -24439.827,E2 -24439.827} C_VEL
LIN {X 0,Y 185.628,Z 656.254,A -85,B 0,C 180,E1 -24440.387,E2 -24440.387} C_VEL
LIN {X 0,Y 187.386,Z 630.665,A -85,B 0,C 180,E1 -24441.237,E2 -24441.237} C_VEL
LIN {X 0,Y 182.68,Z 619.88,A -85,B 0,C 180,E1 -24443.65,E2 -24443.65} C_VEL
LIN {X 0,Y 176.518,Z 609.378,A -85,B 0,C 180,E1 -24446.988,E2 -24446.988} C_VEL
LIN {X 0,Y 171.183,Z 601.37,A -85,B 0,C 180,E1 -24450.256,E2 -24450.256} C_VEL
LIN {X 0,Y 168.201,Z 597.159,A -85,B 0,C 180,E1 -24452.3,E2 -24452.3} C_VEL
LIN {X 0,Y 165.394,Z 593.282,A -85,B 0,C 180,E1 -24454.415,E2 -24454.415} C_VEL
LIN {X 0,Y 162.678,Z 589.506,A -85,B 0,C 180,E1 -24456.698,E2 -24456.698} C_VEL
LIN {X 0,Y 159.345,Z 585.616,A -85,B 0,C 180,E1 -24459.835,E2 -24459.835} C_VEL
LIN {X 0,Y 158.511,Z 584.068,A -85,B 0,C 180,E1 -24460.783,E2 -24460.783} C_VEL
LIN {X 0,Y 155.992,Z 581.868,A -85,B 0,C 180,E1 -24463.645,E2 -24463.645} C_VEL
LIN {X 0,Y 154.322,Z 578.648,A -85,B 0,C 180,E1 -24466.167,E2 -24466.167} C_VEL
LIN {X 0,Y 151.245,Z 576.395,A -85,B 0,C 180,E1 -24471.65,E2 -24471.65} C_VEL
LIN {X 0,Y 149.903,Z 573.592,A -85,B 0,C 180,E1 -24476.304,E2 -24476.304} C_VEL
LIN {X 0,Y 149.783,Z 572.685,A -85,B 0,C 180,E1 -24477.31,E2 -24477.31} C_VEL
LIN {X 0,Y 149.344,Z 572.604,A -85,B 0,C 180,E1 -24482.697,E2 -24482.697} C_VEL
LIN {X 0,Y 149.766,Z 572.936,A -85,B 0,C 180,E1 -24486.399,E2 -24486.399} C_VEL
LIN {X 0,Y 151.42,Z 576.793,A -85,B 0,C 180,E1 -24492.458,E2 -24492.458} C_VEL
LIN {X 0,Y 154.408,Z 578.911,A -85,B 0,C 180,E1 -24497.636,E2 -24497.636} C_VEL
LIN {X 0,Y 155.804,Z 581.755,A -85,B 0,C 180,E1 -24499.774,E2 -24499.774} C_VEL
LIN {X 0,Y 158.474,Z 584.107,A -85,B 0,C 180,E1 -24502.833,E2 -24502.833} C_VEL
LIN {X 0,Y 161.216,Z 588.135,A -85,B 0,C 180,E1 -24505.671,E2 -24505.671} C_VEL
LIN {X 0,Y 162.816,Z 589.751,A -85,B 0,C 180,E1 -24507.076,E2 -24507.076} C_VEL
LIN {X 0,Y 166.391,Z 594.771,A -85,B 0,C 180,E1 -24510.017,E2 -24510.017} C_VEL
LIN {X 0,Y 170.087,Z 600.98,A -85,B 0,C 180,E1 -24512.754,E2 -24512.754} C_VEL
LIN {X 0,Y 174.044,Z 607.912,A -85,B 0,C 180,E1 -24515.366,E2 -24515.366} C_VEL
LIN {X 0,Y 179.701,Z 619.309,A -85,B 0,C 180,E1 -24518.737,E2 -24518.737} C_VEL
LIN {X 0,Y 184.22,Z 629.808,A -85,B 0,C 180,E1 -24521.198,E2 -24521.198} C_VEL
LIN {X 0,Y 186.966,Z 637.173,A -85,B 0,C 180,E1 -24522.634,E2 -24522.634} C_VEL
LIN {X 0,Y 184.282,Z 673.38,A -85,B 0,C 180,E1 -24523.871,E2 -24523.871} C_VEL
LIN {X 0,Y 182.205,Z 687.019,A -85,B 0,C 180,E1 -24524.67,E2 -24524.67} C_VEL
LIN {X 0,Y 179.424,Z 699.383,A -85,B 0,C 180,E1 -24525.758,E2 -24525.758} C_VEL
LIN {X 0,Y 175.765,Z 711.229,A -85,B 0,C 180,E1 -24527.177,E2 -24527.177} C_VEL
LIN {X 0,Y 171.543,Z 722.615,A -85,B 0,C 180,E1 -24529.043,E2 -24529.043} C_VEL
LIN {X 0,Y 167.093,Z 732.891,A -85,B 0,C 180,E1 -24531.271,E2 -24531.271} C_VEL
LIN {X 0,Y 161.995,Z 742.941,A -85,B 0,C 180,E1 -24534.15,E2 -24534.15} C_VEL
LIN {X 0,Y 156.959,Z 751.784,A -85,B 0,C 180,E1 -24537.5,E2 -24537.5} C_VEL
LIN {X 0,Y 152.798,Z 758.604,A -85,B 0,C 180,E1 -24540.916,E2 -24540.916} C_VEL
LIN {X 0,Y 148.935,Z 764.58,A -85,B 0,C 180,E1 -24544.869,E2 -24544.869} C_VEL
LIN {X 0,Y 145.834,Z 769.071,A -85,B 0,C 180,E1 -24548.812,E2 -24548.812} C_VEL
LIN {X 0,Y 143.413,Z 772.493,A -85,B 0,C 180,E1 -24552.901,E2 -24552.901} C_VEL
LIN {X 0,Y 141.63,Z 775.17,A -85,B 0,C 180,E1 -24557.786,E2 -24557.786} C_VEL
LIN {X 0,Y 140.476,Z 776.097,A -85,B 0,C 180,E1 -24560.107,E2 -24560.107} C_VEL
LIN {X 0,Y 137.261,Z 776.903,A -85,B 0,C 180,E1 -24563.953,E2 -24563.953} C_VEL
LIN {X 0,Y 134.74,Z 776.931,A -85,B 0,C 180,E1 -24567.153,E2 -24567.153} C_VEL
LIN {X 0,Y 133.495,Z 776.414,A -85,B 0,C 180,E1 -24570.505,E2 -24570.505} C_VEL
LIN {X 0,Y 133.466,Z 775.831,A -85,B 0,C 180,E1 -24573.018,E2 -24573.018} C_VEL
LIN {X 0,Y 133.539,Z 774.707,A -85,B 0,C 180,E1 -24576.042,E2 -24576.042} C_VEL
LIN {X 0,Y 133.82,Z 773.139,A -85,B 0,C 180,E1 -24579.065,E2 -24579.065} C_VEL
LIN {X 0,Y 134.782,Z 769.989,A -85,B 0,C 180,E1 -24583.57,E2 -24583.57} C_VEL
LIN {X 0,Y 136.393,Z 765.769,A -85,B 0,C 180,E1 -24588.009,E2 -24588.009} C_VEL
LIN {X 0,Y 139.42,Z 759.358,A -85,B 0,C 180,E1 -24592.996,E2 -24592.996} C_VEL
LIN {X 0,Y 142.775,Z 752.265,A -85,B 0,C 180,E1 -24597.144,E2 -24597.144} C_VEL
LIN {X 0,Y 146.518,Z 743.574,A -85,B 0,C 180,E1 -24601.04,E2 -24601.04} C_VEL
LIN {X 0,Y 150.687,Z 733.599,A -85,B 0,C 180,E1 -24604.436,E2 -24604.436} C_VEL
LIN {X 0,Y 154.548,Z 723.458,A -85,B 0,C 180,E1 -24607.051,E2 -24607.051} C_VEL
LIN {X 0,Y 158.177,Z 712.175,A -85,B 0,C 180,E1 -24609.281,E2 -24609.281} C_VEL
LIN {X 0,Y 161.594,Z 699.489,A -85,B 0,C 180,E1 -24611.132,E2 -24611.132} C_VEL
LIN {X 0,Y 164.126,Z 687.076,A -85,B 0,C 180,E1 -24612.408,E2 -24612.408} C_VEL
LIN {X 0,Y 166.062,Z 673.559,A -85,B 0,C 180,E1 -24613.315,E2 -24613.315} C_VEL
LIN {X 0,Y 169.023,Z 629.162,A -85,B 0,C 180,E1 -24615.02,E2 -24615.02} C_VEL
LIN {X 0,Y 168.685,Z 625.665,A -85,B 0,C 180,E1 -24615.326,E2 -24615.326} C_VEL
LIN {X 0,Y 163.978,Z 612.835,A -85,B 0,C 180,E1 -24617.672,E2 -24617.672} C_VEL
LIN {X 0,Y 158.903,Z 601.615,A -85,B 0,C 180,E1 -24620.309,E2 -24620.309} C_VEL
LIN {X 0,Y 153.258,Z 590.858,A -85,B 0,C 180,E1 -24623.508,E2 -24623.508} C_VEL
LIN {X 0,Y 150.137,Z 586.431,A -85,B 0,C 180,E1 -24625.368,E2 -24625.368} C_VEL
LIN {X 0,Y 147.593,Z 582.844,A -85,B 0,C 180,E1 -24627.006,E2 -24627.006} C_VEL
LIN {X 0,Y 145.081,Z 579.675,A -85,B 0,C 180,E1 -24628.719,E2 -24628.719} C_VEL
LIN {X 0,Y 144.156,Z 578.208,A -85,B 0,C 180,E1 -24629.412,E2 -24629.412} C_VEL
LIN {X 0,Y 141.65,Z 575.63,A -85,B 0,C 180,E1 -24631.273,E2 -24631.273} C_VEL
LIN {X 0,Y 140.181,Z 573.053,A -85,B 0,C 180,E1 -24632.552,E2 -24632.552} C_VEL
LIN {X 0,Y 137.727,Z 571.237,A -85,B 0,C 180,E1 -24634.599,E2 -24634.599} C_VEL
LIN {X 0,Y 136.416,Z 568.927,A -85,B 0,C 180,E1 -24635.941,E2 -24635.941} C_VEL
LIN {X 0,Y 136.106,Z 567.518,A -85,B 0,C 180,E1 -24636.443,E2 -24636.443} C_VEL
LIN {X 0,Y 136.239,Z 567.51,A -85,B 0,C 180,E1 -24638.832,E2 -24638.832} C_VEL
LIN {X 0,Y 136.268,Z 567.51,A -85,B 0,C 180,E1 -24645.056,E2 -24645.056} C_VEL
LIN {X 0,Y 136.495,Z 567.466,A -85,B 0,C 180,E1 -24648.115,E2 -24648.115} C_VEL
LIN {X 0,Y 136.586,Z 567.468,A -85,B 0,C 180,E1 -24651.12,E2 -24651.12} C_VEL
LIN {X 0,Y 137.13,Z 567.399,A -85,B 0,C 180,E1 -24660,E2 -24660} C_VEL
LIN {X 0,Y 136.55,Z 567.45,A -85,B 0,C 180,E1 -24668.883,E2 -24668.883} C_VEL
LIN {X 0,Y 136.438,Z 567.457,A -85,B 0,C 180,E1 -24671.891,E2 -24671.891} C_VEL
LIN {X 0,Y 136.208,Z 567.495,A -85,B 0,C 180,E1 -24678.035,E2 -24678.035} C_VEL
LIN {X 0,Y 136.196,Z 567.496,A -85,B 0,C 180,E1 -24681.749,E2 -24681.749} C_VEL
LIN {X 0,Y 136.135,Z 567.521,A -85,B 0,C 180,E1 -24688.094,E2 -24688.094} C_VEL
LIN {X 0,Y 136.841,Z 569.912,A -85,B 0,C 180,E1 -24688.988,E2 -24688.988} C_VEL
LIN {X 0,Y 138.637,Z 572.182,A -85,B 0,C 180,E1 -24690.671,E2 -24690.671} C_VEL
LIN {X 0,Y 140.538,Z 573.462,A -85,B 0,C 180,E1 -24692.202,E2 -24692.202} C_VEL
LIN {X 0,Y 142.411,Z 576.658,A -85,B 0,C 180,E1 -24693.79,E2 -24693.79} C_VEL
LIN {X 0,Y 144.588,Z 578.787,A -85,B 0,C 180,E1 -24695.362,E2 -24695.362} C_VEL
LIN {X 0,Y 147.332,Z 582.593,A -85,B 0,C 180,E1 -24697.285,E2 -24697.285} C_VEL
LIN {X 0,Y 151.997,Z 589.104,A -85,B 0,C 180,E1 -24700.219,E2 -24700.219} C_VEL
LIN {X 0,Y 156.962,Z 596.437,A -85,B 0,C 180,E1 -24702.996,E2 -24702.996} C_VEL
LIN {X 0,Y 163.098,Z 606.896,A -85,B 0,C 180,E1 -24706.1,E2 -24706.1} C_VEL
LIN {X 0,Y 168.279,Z 617.269,A -85,B 0,C 180,E1 -24708.517,E2 -24708.517} C_VEL
LIN {X 0,Y 169.575,Z 620.735,A -85,B 0,C 180,E1 -24709.133,E2 -24709.133} C_VEL
LIN {X 0,Y 166.506,Z 665.895,A -85,B 0,C 180,E1 -24710.829,E2 -24710.829} C_VEL
LIN {X 0,Y 164.789,Z 678.947,A -85,B 0,C 180,E1 -24711.718,E2 -24711.718} C_VEL
LIN {X 0,Y 162.354,Z 691.989,A -85,B 0,C 180,E1 -24713.087,E2 -24713.087} C_VEL
LIN {X 0,Y 159.479,Z 703.068,A -85,B 0,C 180,E1 -24714.663,E2 -24714.663} C_VEL
LIN {X 0,Y 156.498,Z 713.278,A -85,B 0,C 180,E1 -24716.626,E2 -24716.626} C_VEL
LIN {X 0,Y 152.777,Z 723.855,A -85,B 0,C 180,E1 -24719.219,E2 -24719.219} C_VEL
LIN {X 0,Y 148.417,Z 734.261,A -85,B 0,C 180,E1 -24722.504,E2 -24722.504} C_VEL
LIN {X 0,Y 145.029,Z 741.91,A -85,B 0,C 180,E1 -24725.676,E2 -24725.676} C_VEL
LIN {X 0,Y 141.653,Z 749.392,A -85,B 0,C 180,E1 -24729.678,E2 -24729.678} C_VEL
LIN {X 0,Y 138.821,Z 755.412,A -85,B 0,C 180,E1 -24733.833,E2 -24733.833} C_VEL
LIN {X 0,Y 136.547,Z 760.187,A -85,B 0,C 180,E1 -24738.119,E2 -24738.119} C_VEL
LIN {X 0,Y 134.958,Z 763.768,A -85,B 0,C 180,E1 -24742.389,E2 -24742.389} C_VEL
LIN {X 0,Y 133.922,Z 766.526,A -85,B 0,C 180,E1 -24746.992,E2 -24746.992} C_VEL
LIN {X 0,Y 133.543,Z 768.033,A -85,B 0,C 180,E1 -24750.678,E2 -24750.678} C_VEL
LIN {X 0,Y 133.465,Z 769.105,A -85,B 0,C 180,E1 -24756.045,E2 -24756.045} C_VEL
LIN {X 0,Y 133.694,Z 769.161,A -85,B 0,C 180,E1 -24759.073,E2 -24759.073} C_VEL
LIN {X 0,Y 134.165,Z 768.837,A -85,B 0,C 180,E1 -24762.095,E2 -24762.095} C_VEL
LIN {X 0,Y 134.877,Z 768.13,A -85,B 0,C 180,E1 -24765.101,E2 -24765.101} C_VEL
LIN {X 0,Y 135.922,Z 766.985,A -85,B 0,C 180,E1 -24768.073,E2 -24768.073} C_VEL
LIN {X 0,Y 137.303,Z 765.422,A -85,B 0,C 180,E1 -24770.995,E2 -24770.995} C_VEL
LIN {X 0,Y 139.863,Z 762.305,A -85,B 0,C 180,E1 -24775.244,E2 -24775.244} C_VEL
LIN {X 0,Y 143.161,Z 758.055,A -85,B 0,C 180,E1 -24779.4,E2 -24779.4} C_VEL
LIN {X 0,Y 147.803,Z 751.634,A -85,B 0,C 180,E1 -24783.966,E2 -24783.966} C_VEL
LIN {X 0,Y 152.537,Z 744.576,A -85,B 0,C 180,E1 -24787.623,E2 -24787.623} C_VEL
LIN {X 0,Y 157.573,Z 735.905,A -85,B 0,C 180,E1 -24791.052,E2 -24791.052} C_VEL
LIN {X 0,Y 162.424,Z 726.668,A -85,B 0,C 180,E1 -24793.812,E2 -24793.812} C_VEL
LIN {X 0,Y 167.016,Z 716.623,A -85,B 0,C 180,E1 -24796.104,E2 -24796.104} C_VEL
LIN {X 0,Y 171.338,Z 705.423,A -85,B 0,C 180,E1 -24798.025,E2 -24798.025} C_VEL
LIN {X 0,Y 174.523,Z 694.82,A -85,B 0,C 180,E1 -24799.471,E2 -24799.471} C_VEL
LIN {X 0,Y 177.529,Z 682.351,A -85,B 0,C 180,E1 -24800.697,E2 -24800.697} C_VEL
LIN {X 0,Y 179.711,Z 669.195,A -85,B 0,C 180,E1 -24801.568,E2 -24801.568} C_VEL
LIN {X 0,Y 181.368,Z 651.457,A -85,B 0,C 180,E1 -24802.22,E2 -24802.22} C_VEL
LIN {X 0,Y 182.605,Z 633.017,A -85,B 0,C 180,E1 -24802.87,E2 -24802.87} C_VEL
LIN {X 0,Y 178.794,Z 624.265,A -85,B 0,C 180,E1 -24804.97,E2 -24804.97} C_VEL
LIN {X 0,Y 173.266,Z 614.587,A -85,B 0,C 180,E1 -24808.176,E2 -24808.176} C_VEL
LIN {X 0,Y 168.467,Z 607.163,A -85,B 0,C 180,E1 -24811.309,E2 -24811.309} C_VEL
LIN {X 0,Y 165.454,Z 602.758,A -85,B 0,C 180,E1 -24813.515,E2 -24813.515} C_VEL
LIN {X 0,Y 163.08,Z 599.343,A -85,B 0,C 180,E1 -24815.43,E2 -24815.43} C_VEL
LIN {X 0,Y 160.129,Z 595.309,A -85,B 0,C 180,E1 -24818.074,E2 -24818.074} C_VEL
LIN {X 0,Y 157.31,Z 591.65,A -85,B 0,C 180,E1 -24820.975,E2 -24820.975} C_VEL
LIN {X 0,Y 156.696,Z 590.647,A -85,B 0,C 180,E1 -24821.702,E2 -24821.702} C_VEL
LIN {X 0,Y 154.166,Z 588.015,A -85,B 0,C 180,E1 -24824.846,E2 -24824.846} C_VEL
LIN {X 0,Y 152.83,Z 585.442,A -85,B 0,C 180,E1 -24827.024,E2 -24827.024} C_VEL
LIN {X 0,Y 149.994,Z 583.012,A -85,B 0,C 180,E1 -24832.596,E2 -24832.596} C_VEL
LIN {X 0,Y 148.887,Z 580.276,A -85,B 0,C 180,E1 -24837.125,E2 -24837.125} C_VEL
LIN {X 0,Y 148.796,Z 579.673,A -85,B 0,C 180,E1 -24837.97,E2 -24837.97} C_VEL
LIN {X 0,Y 148.843,Z 579.931,A -85,B 0,C 180,E1 -24846.098,E2 -24846.098} C_VEL
LIN {X 0,Y 149.887,Z 583.068,A -85,B 0,C 180,E1 -24850.81,E2 -24850.81} C_VEL
LIN {X 0,Y 152.453,Z 585.339,A -85,B 0,C 180,E1 -24856.057,E2 -24856.057} C_VEL
LIN {X 0,Y 153.002,Z 585.818,A -85,B 0,C 180,E1 -24856.929,E2 -24856.929} C_VEL
LIN {X 0,Y 154.823,Z 589.065,A -85,B 0,C 180,E1 -24859.731,E2 -24859.731} C_VEL
LIN {X 0,Y 157.099,Z 591.241,A -85,B 0,C 180,E1 -24862.416,E2 -24862.416} C_VEL
LIN {X 0,Y 159.435,Z 594.687,A -85,B 0,C 180,E1 -24864.93,E2 -24864.93} C_VEL
LIN {X 0,Y 160.889,Z 596.281,A -85,B 0,C 180,E1 -24866.281,E2 -24866.281} C_VEL
LIN {X 0,Y 164.006,Z 600.806,A -85,B 0,C 180,E1 -24868.997,E2 -24868.997} C_VEL
LIN {X 0,Y 168.805,Z 609.123,A -85,B 0,C 180,E1 -24872.689,E2 -24872.689} C_VEL
LIN {X 0,Y 173.227,Z 617.87,A -85,B 0,C 180,E1 -24875.69,E2 -24875.69} C_VEL
LIN {X 0,Y 177.98,Z 628.332,A -85,B 0,C 180,E1 -24878.595,E2 -24878.595} C_VEL
LIN {X 0,Y 182.224,Z 639.486,A -85,B 0,C 180,E1 -24881.024,E2 -24881.024} C_VEL
LIN {X 0,Y 179.582,Z 673.526,A -85,B 0,C 180,E1 -24882.208,E2 -24882.208} C_VEL
LIN {X 0,Y 177.383,Z 687.253,A -85,B 0,C 180,E1 -24883.019,E2 -24883.019} C_VEL
LIN {X 0,Y 174.429,Z 699.726,A -85,B 0,C 180,E1 -24884.137,E2 -24884.137} C_VEL
LIN {X 0,Y 170.649,Z 711.452,A -85,B 0,C 180,E1 -24885.564,E2 -24885.564} C_VEL
LIN {X 0,Y 166.257,Z 722.76,A -85,B 0,C 180,E1 -24887.442,E2 -24887.442} C_VEL
LIN {X 0,Y 161.623,Z 732.963,A -85,B 0,C 180,E1 -24889.699,E2 -24889.699} C_VEL
LIN {X 0,Y 156.279,Z 742.956,A -85,B 0,C 180,E1 -24892.621,E2 -24892.621} C_VEL
LIN {X 0,Y 151.019,Z 751.762,A -85,B 0,C 180,E1 -24896.052,E2 -24896.052} C_VEL
LIN {X 0,Y 146.303,Z 758.999,A -85,B 0,C 180,E1 -24899.845,E2 -24899.845} C_VEL
LIN {X 0,Y 142.528,Z 764.483,A -85,B 0,C 180,E1 -24903.655,E2 -24903.655} C_VEL
LIN {X 0,Y 139.218,Z 768.949,A -85,B 0,C 180,E1 -24907.753,E2 -24907.753} C_VEL
LIN {X 0,Y 136.609,Z 772.347,A -85,B 0,C 180,E1 -24912.021,E2 -24912.021} C_VEL
LIN {X 0,Y 134.472,Z 775.348,A -85,B 0,C 180,E1 -24917.933,E2 -24917.933} C_VEL
LIN {X 0,Y 133.839,Z 776.26,A -85,B 0,C 180,E1 -24920.936,E2 -24920.936} C_VEL
LIN {X 0,Y 133.502,Z 776.751,A -85,B 0,C 180,E1 -24923.956,E2 -24923.956} C_VEL
LIN {X 0,Y 133.407,Z 776.833,A -85,B 0,C 180,E1 -24926.98,E2 -24926.98} C_VEL
LIN {X 0,Y 133.495,Z 776.414,A -85,B 0,C 180,E1 -24930.505,E2 -24930.505} C_VEL
LIN {X 0,Y 132.736,Z 775.814,A -85,B 0,C 180,E1 -24933.007,E2 -24933.007} C_VEL
LIN {X 0,Y 130.025,Z 774.153,A -85,B 0,C 180,E1 -24937.109,E2 -24937.109} C_VEL
LIN {X 0,Y 128.045,Z 772.359,A -85,B 0,C 180,E1 -24940.46,E2 -24940.46} C_VEL
LIN {X 0,Y 127.565,Z 770.689,A -85,B 0,C 180,E1 -24943.016,E2 -24943.016} C_VEL
LIN {X 0,Y 127.714,Z 770.043,A -85,B 0,C 180,E1 -24943.862,E2 -24943.862} C_VEL
LIN {X 0,Y 129.629,Z 765.454,A -85,B 0,C 180,E1 -24948.983,E2 -24948.983} C_VEL
LIN {X 0,Y 132.847,Z 759.014,A -85,B 0,C 180,E1 -24954.204,E2 -24954.204} C_VEL
LIN {X 0,Y 136.278,Z 752.234,A -85,B 0,C 180,E1 -24958.328,E2 -24958.328} C_VEL
LIN {X 0,Y 140.437,Z 743.146,A -85,B 0,C 180,E1 -24962.545,E2 -24962.545} C_VEL
LIN {X 0,Y 144.861,Z 733.127,A -85,B 0,C 180,E1 -24966.032,E2 -24966.032} C_VEL
LIN {X 0,Y 148.925,Z 722.901,A -85,B 0,C 180,E1 -24968.702,E2 -24968.702} C_VEL
LIN {X 0,Y 152.734,Z 711.54,A -85,B 0,C 180,E1 -24970.972,E2 -24970.972} C_VEL
LIN {X 0,Y 156.042,Z 699.748,A -85,B 0,C 180,E1 -24972.718,E2 -24972.718} C_VEL
LIN {X 0,Y 158.679,Z 687.572,A -85,B 0,C 180,E1 -24974.011,E2 -24974.011} C_VEL
LIN {X 0,Y 160.725,Z 674.11,A -85,B 0,C 180,E1 -24974.943,E2 -24974.943} C_VEL
LIN {X 0,Y 162.797,Z 646.216,A -85,B 0,C 180,E1 -24976.058,E2 -24976.058} C_VEL
LIN {X 0,Y 163.817,Z 629.513,A -85,B 0,C 180,E1 -24976.714,E2 -24976.714} C_VEL
LIN {X 0,Y 163.157,Z 626.79,A -85,B 0,C 180,E1 -24977.109,E2 -24977.109} C_VEL
LIN {X 0,Y 158.638,Z 614.466,A -85,B 0,C 180,E1 -24979.566,E2 -24979.566} C_VEL
LIN {X 0,Y 153.581,Z 603.41,A -85,B 0,C 180,E1 -24982.448,E2 -24982.448} C_VEL
LIN {X 0,Y 149.373,Z 595.477,A -85,B 0,C 180,E1 -24985.05,E2 -24985.05} C_VEL
LIN {X 0,Y 144.856,Z 588.826,A -85,B 0,C 180,E1 -24988.053,E2 -24988.053} C_VEL
LIN {X 0,Y 142.158,Z 585.232,A -85,B 0,C 180,E1 -24990.027,E2 -24990.027} C_VEL
LIN {X 0,Y 140.88,Z 583.74,A -85,B 0,C 180,E1 -24991.008,E2 -24991.008} C_VEL
LIN {X 0,Y 138.567,Z 580.694,A -85,B 0,C 180,E1 -24992.943,E2 -24992.943} C_VEL
LIN {X 0,Y 137.752,Z 579.422,A -85,B 0,C 180,E1 -24993.69,E2 -24993.69} C_VEL
LIN {X 0,Y 135.278,Z 577.136,A -85,B 0,C 180,E1 -24995.952,E2 -24995.952} C_VEL
LIN {X 0,Y 133.621,Z 574.14,A -85,B 0,C 180,E1 -24997.813,E2 -24997.813} C_VEL
LIN {X 0,Y 130.806,Z 572.149,A -85,B 0,C 180,E1 -25000.991,E2 -25000.991} C_VEL
LIN {X 0,Y 129.375,Z 569.508,A -85,B 0,C 180,E1 -25003.125,E2 -25003.125} C_VEL
LIN {X 0,Y 129.169,Z 568.382,A -85,B 0,C 180,E1 -25003.707,E2 -25003.707} C_VEL
LIN {X 0,Y 129.414,Z 568.348,A -85,B 0,C 180,E1 -25007.821,E2 -25007.821} C_VEL
LIN {X 0,Y 129.512,Z 568.343,A -85,B 0,C 180,E1 -25010.631,E2 -25010.631} C_VEL
LIN {X 0,Y 130.085,Z 568.276,A -85,B 0,C 180,E1 -25020,E2 -25020} C_VEL
LIN {X 0,Y 129.472,Z 568.326,A -85,B 0,C 180,E1 -25029.373,E2 -25029.373} C_VEL
LIN {X 0,Y 129.342,Z 568.344,A -85,B 0,C 180,E1 -25032.554,E2 -25032.554} C_VEL
LIN {X 0,Y 129.129,Z 568.369,A -85,B 0,C 180,E1 -25039.06,E2 -25039.06} C_VEL
LIN {X 0,Y 129.208,Z 568.436,A -85,B 0,C 180,E1 -25040.933,E2 -25040.933} C_VEL
LIN {X 0,Y 129.932,Z 570.896,A -85,B 0,C 180,E1 -25042.249,E2 -25042.249} C_VEL
LIN {X 0,Y 131.74,Z 573.157,A -85,B 0,C 180,E1 -25044.632,E2 -25044.632} C_VEL
LIN {X 0,Y 133.905,Z 574.454,A -85,B 0,C 180,E1 -25046.95,E2 -25046.95} C_VEL
LIN {X 0,Y 135.425,Z 577.378,A -85,B 0,C 180,E1 -25048.659,E2 -25048.659} C_VEL
LIN {X 0,Y 137.662,Z 579.434,A -85,B 0,C 180,E1 -25050.7,E2 -25050.7} C_VEL
LIN {X 0,Y 138.301,Z 580.145,A -85,B 0,C 180,E1 -25051.26,E2 -25051.26} C_VEL
LIN {X 0,Y 140.714,Z 583.626,A -85,B 0,C 180,E1 -25053.326,E2 -25053.326} C_VEL
LIN {X 0,Y 142.175,Z 585.285,A -85,B 0,C 180,E1 -25054.446,E2 -25054.446} C_VEL
LIN {X 0,Y 145.835,Z 590.436,A -85,B 0,C 180,E1 -25057.105,E2 -25057.105} C_VEL
LIN {X 0,Y 150.489,Z 597.079,A -85,B 0,C 180,E1 -25060.089,E2 -25060.089} C_VEL
LIN {X 0,Y 156.01,Z 606.069,A -85,B 0,C 180,E1 -25063.255,E2 -25063.255} C_VEL
LIN {X 0,Y 161.616,Z 616.629,A -85,B 0,C 180,E1 -25066.164,E2 -25066.164} C_VEL
LIN {X 0,Y 164.318,Z 622.804,A -85,B 0,C 180,E1 -25067.512,E2 -25067.512} C_VEL
LIN {X 0,Y 161.253,Z 666.178,A -85,B 0,C 180,E1 -25069.176,E2 -25069.176} C_VEL
LIN {X 0,Y 159.42,Z 679.366,A -85,B 0,C 180,E1 -25070.084,E2 -25070.084} C_VEL
LIN {X 0,Y 157.015,Z 691.754,A -85,B 0,C 180,E1 -25071.404,E2 -25071.404} C_VEL
LIN {X 0,Y 153.771,Z 703.743,A -85,B 0,C 180,E1 -25073.14,E2 -25073.14} C_VEL
LIN {X 0,Y 150.64,Z 713.867,A -85,B 0,C 180,E1 -25075.145,E2 -25075.145} C_VEL
LIN {X 0,Y 146.75,Z 724.378,A -85,B 0,C 180,E1 -25077.807,E2 -25077.807} C_VEL
LIN {X 0,Y 142.958,Z 732.986,A -85,B 0,C 180,E1 -25080.554,E2 -25080.554} C_VEL
LIN {X 0,Y 139.223,Z 740.907,A -85,B 0,C 180,E1 -25083.788,E2 -25083.788} C_VEL
LIN {X 0,Y 135.595,Z 748.654,A -85,B 0,C 180,E1 -25087.929,E2 -25087.929} C_VEL
LIN {X 0,Y 132.034,Z 755.751,A -85,B 0,C 180,E1 -25092.977,E2 -25092.977} C_VEL
LIN {X 0,Y 129.63,Z 760.498,A -85,B 0,C 180,E1 -25097.475,E2 -25097.475} C_VEL
LIN {X 0,Y 127.893,Z 764.144,A -85,B 0,C 180,E1 -25102.104,E2 -25102.104} C_VEL
LIN {X 0,Y 126.835,Z 766.785,A -85,B 0,C 180,E1 -25106.824,E2 -25106.824} C_VEL
LIN {X 0,Y 126.506,Z 768.033,A -85,B 0,C 180,E1 -25110,E2 -25110} C_VEL
LIN {X 0,Y 126.384,Z 768.887,A -85,B 0,C 180,E1 -25113.188,E2 -25113.188} C_VEL
LIN {X 0,Y 126.398,Z 769.316,A -85,B 0,C 180,E1 -25116.385,E2 -25116.385} C_VEL
LIN {X 0,Y 127.2,Z 769.025,A -85,B 0,C 180,E1 -25122.768,E2 -25122.768} C_VEL
LIN {X 0,Y 127.975,Z 768.302,A -85,B 0,C 180,E1 -25125.937,E2 -25125.937} C_VEL
LIN {X 0,Y 129.154,Z 767.136,A -85,B 0,C 180,E1 -25129.056,E2 -25129.056} C_VEL
LIN {X 0,Y 130.634,Z 765.562,A -85,B 0,C 180,E1 -25132.122,E2 -25132.122} C_VEL
LIN {X 0,Y 133.136,Z 762.738,A -85,B 0,C 180,E1 -25136.181,E2 -25136.181} C_VEL
LIN {X 0,Y 136.974,Z 758.14,A -85,B 0,C 180,E1 -25140.869,E2 -25140.869} C_VEL
LIN {X 0,Y 141.932,Z 751.686,A -85,B 0,C 180,E1 -25145.578,E2 -25145.578} C_VEL
LIN {X 0,Y 146.926,Z 744.583,A -85,B 0,C 180,E1 -25149.326,E2 -25149.326} C_VEL
LIN {X 0,Y 152.352,Z 735.705,A -85,B 0,C 180,E1 -25152.874,E2 -25152.874} C_VEL
LIN {X 0,Y 157.322,Z 726.58,A -85,B 0,C 180,E1 -25155.623,E2 -25155.623} C_VEL
LIN {X 0,Y 162.162,Z 716.44,A -85,B 0,C 180,E1 -25157.917,E2 -25157.917} C_VEL
LIN {X 0,Y 166.635,Z 705.151,A -85,B 0,C 180,E1 -25159.856,E2 -25159.856} C_VEL
LIN {X 0,Y 170.265,Z 693.43,A -85,B 0,C 180,E1 -25161.413,E2 -25161.413} C_VEL
LIN {X 0,Y 173.284,Z 680.758,A -85,B 0,C 180,E1 -25162.602,E2 -25162.602} C_VEL
LIN {X 0,Y 175.401,Z 668.035,A -85,B 0,C 180,E1 -25163.379,E2 -25163.379} C_VEL
LIN {X 0,Y 177.335,Z 645.894,A -85,B 0,C 180,E1 -25164.176,E2 -25164.176} C_VEL
LIN {X 0,Y 178.009,Z 635.507,A -85,B 0,C 180,E1 -25164.568,E2 -25164.568} C_VEL
LIN {X 0,Y 175.112,Z 628.89,A -85,B 0,C 180,E1 -25166.283,E2 -25166.283} C_VEL
LIN {X 0,Y 170.279,Z 620.133,A -85,B 0,C 180,E1 -25169.285,E2 -25169.285} C_VEL
LIN {X 0,Y 165.916,Z 613.1,A -85,B 0,C 180,E1 -25172.32,E2 -25172.32} C_VEL
LIN {X 0,Y 162.846,Z 608.442,A -85,B 0,C 180,E1 -25174.721,E2 -25174.721} C_VEL
LIN {X 0,Y 160.787,Z 605.437,A -85,B 0,C 180,E1 -25176.493,E2 -25176.493} C_VEL
LIN {X 0,Y 158.15,Z 601.656,A -85,B 0,C 180,E1 -25179.017,E2 -25179.017} C_VEL
LIN {X 0,Y 155.362,Z 597.727,A -85,B 0,C 180,E1 -25182.114,E2 -25182.114} C_VEL
LIN {X 0,Y 152.362,Z 594.083,A -85,B 0,C 180,E1 -25186.155,E2 -25186.155} C_VEL
LIN {X 0,Y 151.587,Z 592.357,A -85,B 0,C 180,E1 -25187.555,E2 -25187.555} C_VEL
LIN {X 0,Y 148.783,Z 589.646,A -85,B 0,C 180,E1 -25193.558,E2 -25193.558} C_VEL
LIN {X 0,Y 147.889,Z 586.823,A -85,B 0,C 180,E1 -25198.127,E2 -25198.127} C_VEL
LIN {X 0,Y 147.613,Z 586.701,A -85,B 0,C 180,E1 -25202.729,E2 -25202.729} C_VEL
LIN {X 0,Y 147.911,Z 587.034,A -85,B 0,C 180,E1 -25205.795,E2 -25205.795} C_VEL
LIN {X 0,Y 149.288,Z 590.65,A -85,B 0,C 180,E1 -25211.609,E2 -25211.609} C_VEL
LIN {X 0,Y 151.649,Z 592.671,A -85,B 0,C 180,E1 -25216.241,E2 -25216.241} C_VEL
LIN {X 0,Y 153.494,Z 595.919,A -85,B 0,C 180,E1 -25219.213,E2 -25219.213} C_VEL
LIN {X 0,Y 155.462,Z 597.911,A -85,B 0,C 180,E1 -25221.657,E2 -25221.657} C_VEL
LIN {X 0,Y 157.984,Z 601.547,A -85,B 0,C 180,E1 -25224.473,E2 -25224.473} C_VEL
LIN {X 0,Y 159.198,Z 603.135,A -85,B 0,C 180,E1 -25225.67,E2 -25225.67} C_VEL
LIN {X 0,Y 161.607,Z 606.711,A -85,B 0,C 180,E1 -25227.885,E2 -25227.885} C_VEL
LIN {X 0,Y 165.592,Z 613.974,A -85,B 0,C 180,E1 -25231.203,E2 -25231.203} C_VEL
LIN {X 0,Y 168.775,Z 620.416,A -85,B 0,C 180,E1 -25233.576,E2 -25233.576} C_VEL
LIN {X 0,Y 172.744,Z 629.137,A -85,B 0,C 180,E1 -25236.269,E2 -25236.269} C_VEL
LIN {X 0,Y 176.344,Z 638.194,A -85,B 0,C 180,E1 -25238.542,E2 -25238.542} C_VEL
LIN {X 0,Y 177.634,Z 641.869,A -85,B 0,C 180,E1 -25239.333,E2 -25239.333} C_VEL
LIN {X 0,Y 175.117,Z 672.938,A -85,B 0,C 180,E1 -25240.414,E2 -25240.414} C_VEL
LIN {X 0,Y 172.9,Z 686.452,A -85,B 0,C 180,E1 -25241.196,E2 -25241.196} C_VEL
LIN {X 0,Y 169.876,Z 699.06,A -85,B 0,C 180,E1 -25242.312,E2 -25242.312} C_VEL
LIN {X 0,Y 166.256,Z 710.096,A -85,B 0,C 180,E1 -25243.623,E2 -25243.623} C_VEL
LIN {X 0,Y 162.285,Z 720.323,A -85,B 0,C 180,E1 -25245.274,E2 -25245.274} C_VEL
LIN {X 0,Y 157.355,Z 730.926,A -85,B 0,C 180,E1 -25247.506,E2 -25247.506} C_VEL
LIN {X 0,Y 152.671,Z 739.598,A -85,B 0,C 180,E1 -25249.875,E2 -25249.875} C_VEL
LIN {X 0,Y 147.85,Z 747.592,A -85,B 0,C 180,E1 -25252.695,E2 -25252.695} C_VEL
LIN {X 0,Y 142.642,Z 755.445,A -85,B 0,C 180,E1 -25256.339,E2 -25256.339} C_VEL
LIN {X 0,Y 138.915,Z 760.781,A -85,B 0,C 180,E1 -25259.608,E2 -25259.608} C_VEL
LIN {X 0,Y 134.906,Z 766.007,A -85,B 0,C 180,E1 -25263.717,E2 -25263.717} C_VEL
LIN {X 0,Y 131.632,Z 770.076,A -85,B 0,C 180,E1 -25268.054,E2 -25268.054} C_VEL
LIN {X 0,Y 129.84,Z 772.202,A -85,B 0,C 180,E1 -25271.049,E2 -25271.049} C_VEL
LIN {X 0,Y 128.533,Z 773.891,A -85,B 0,C 180,E1 -25274.134,E2 -25274.134} C_VEL
LIN {X 0,Y 126.808,Z 776.08,A -85,B 0,C 180,E1 -25280.429,E2 -25280.429} C_VEL
LIN {X 0,Y 126.435,Z 776.551,A -85,B 0,C 180,E1 -25283.617,E2 -25283.617} C_VEL
LIN {X 0,Y 126.31,Z 776.623,A -85,B 0,C 180,E1 -25286.81,E2 -25286.81} C_VEL
LIN {X 0,Y 126.415,Z 776.221,A -85,B 0,C 180,E1 -25290.405,E2 -25290.405} C_VEL
LIN {X 0,Y 126.378,Z 775.599,A -85,B 0,C 180,E1 -25293.188,E2 -25293.188} C_VEL
LIN {X 0,Y 126.46,Z 774.452,A -85,B 0,C 180,E1 -25296.381,E2 -25296.381} C_VEL
LIN {X 0,Y 126.785,Z 772.873,A -85,B 0,C 180,E1 -25299.572,E2 -25299.572} C_VEL
LIN {X 0,Y 127.714,Z 770.043,A -85,B 0,C 180,E1 -25303.862,E2 -25303.862} C_VEL
LIN {X 0,Y 127.86,Z 768.065,A -85,B 0,C 180,E1 -25306.363,E2 -25306.363} C_VEL
LIN {X 0,Y 126.759,Z 764.339,A -85,B 0,C 180,E1 -25310.482,E2 -25310.482} C_VEL
LIN {X 0,Y 126.27,Z 759.935,A -85,B 0,C 180,E1 -25314.506,E2 -25314.506} C_VEL
LIN {X 0,Y 127.337,Z 756.895,A -85,B 0,C 180,E1 -25316.744,E2 -25316.744} C_VEL
LIN {X 0,Y 130.96,Z 749.94,A -85,B 0,C 180,E1 -25320.836,E2 -25320.836} C_VEL
LIN {X 0,Y 135.279,Z 741.077,A -85,B 0,C 180,E1 -25324.852,E2 -25324.852} C_VEL
LIN {X 0,Y 140.085,Z 730.508,A -85,B 0,C 180,E1 -25328.377,E2 -25328.377} C_VEL
LIN {X 0,Y 144.388,Z 719.745,A -85,B 0,C 180,E1 -25331.078,E2 -25331.078} C_VEL
LIN {X 0,Y 147.946,Z 709.307,A -85,B 0,C 180,E1 -25333.067,E2 -25333.067} C_VEL
LIN {X 0,Y 151.483,Z 696.758,A -85,B 0,C 180,E1 -25334.798,E2 -25334.798} C_VEL
LIN {X 0,Y 154.097,Z 684.252,A -85,B 0,C 180,E1 -25336.032,E2 -25336.032} C_VEL
LIN {X 0,Y 155.875,Z 671.593,A -85,B 0,C 180,E1 -25336.857,E2 -25336.857} C_VEL
LIN {X 0,Y 158.822,Z 631.16,A -85,B 0,C 180,E1 -25338.413,E2 -25338.413} C_VEL
LIN {X 0,Y 154.73,Z 619.376,A -85,B 0,C 180,E1 -25340.826,E2 -25340.826} C_VEL
LIN {X 0,Y 149.892,Z 608.272,A -85,B 0,C 180,E1 -25343.809,E2 -25343.809} C_VEL
LIN {X 0,Y 146.047,Z 600.783,A -85,B 0,C 180,E1 -25346.371,E2 -25346.371} C_VEL
LIN {X 0,Y 141.837,Z 594.501,A -85,B 0,C 180,E1 -25349.374,E2 -25349.374} C_VEL
LIN {X 0,Y 138.715,Z 590.172,A -85,B 0,C 180,E1 -25351.867,E2 -25351.867} C_VEL
LIN {X 0,Y 136.169,Z 586.804,A -85,B 0,C 180,E1 -25354.12,E2 -25354.12} C_VEL
LIN {X 0,Y 135.269,Z 585.618,A -85,B 0,C 180,E1 -25354.979,E2 -25354.979} C_VEL
LIN {X 0,Y 132.733,Z 582.747,A -85,B 0,C 180,E1 -25357.555,E2 -25357.555} C_VEL
LIN {X 0,Y 131.558,Z 580.69,A -85,B 0,C 180,E1 -25358.974,E2 -25358.974} C_VEL
LIN {X 0,Y 128.981,Z 578.508,A -85,B 0,C 180,E1 -25362.152,E2 -25362.152} C_VEL
LIN {X 0,Y 127.494,Z 575.498,A -85,B 0,C 180,E1 -25364.616,E2 -25364.616} C_VEL
LIN {X 0,Y 123.397,Z 571.994,A -85,B 0,C 180,E1 -25373.46,E2 -25373.46} C_VEL
LIN {X 0,Y 122.724,Z 569.701,A -85,B 0,C 180,E1 -25377.128,E2 -25377.128} C_VEL
LIN {X 0,Y 122.723,Z 569.192,A -85,B 0,C 180,E1 -25377.949,E2 -25377.949} C_VEL
LIN {X 0,Y 123.039,Z 569.152,A -85,B 0,C 180,E1 -25380,E2 -25380} C_VEL
LIN {X 0,Y 122.474,Z 569.29,A -85,B 0,C 180,E1 -25385.351,E2 -25385.351} C_VEL
LIN {X 0,Y 125.021,Z 574.143,A -85,B 0,C 180,E1 -25395.487,E2 -25395.487} C_VEL
LIN {X 0,Y 127.502,Z 575.416,A -85,B 0,C 180,E1 -25399.838,E2 -25399.838} C_VEL
LIN {X 0,Y 128.613,Z 578.083,A -85,B 0,C 180,E1 -25401.779,E2 -25401.779} C_VEL
LIN {X 0,Y 130.747,Z 580.305,A -85,B 0,C 180,E1 -25404.585,E2 -25404.585} C_VEL
LIN {X 0,Y 131.962,Z 581.217,A -85,B 0,C 180,E1 -25405.959,E2 -25405.959} C_VEL
LIN {X 0,Y 134.016,Z 584.514,A -85,B 0,C 180,E1 -25408.286,E2 -25408.286} C_VEL
LIN {X 0,Y 136.025,Z 586.515,A -85,B 0,C 180,E1 -25410.191,E2 -25410.191} C_VEL
LIN {X 0,Y 138.737,Z 590.24,A -85,B 0,C 180,E1 -25412.613,E2 -25412.613} C_VEL
LIN {X 0,Y 142.943,Z 596.182,A -85,B 0,C 180,E1 -25415.915,E2 -25415.915} C_VEL
LIN {X 0,Y 147.386,Z 602.813,A -85,B 0,C 180,E1 -25418.965,E2 -25418.965} C_VEL
LIN {X 0,Y 152.415,Z 611.251,A -85,B 0,C 180,E1 -25422.048,E2 -25422.048} C_VEL
LIN {X 0,Y 157.596,Z 621.39,A -85,B 0,C 180,E1 -25424.936,E2 -25424.936} C_VEL
LIN {X 0,Y 159.221,Z 624.98,A -85,B 0,C 180,E1 -25425.799,E2 -25425.799} C_VEL
LIN {X 0,Y 156.088,Z 666.936,A -85,B 0,C 180,E1 -25427.44,E2 -25427.44} C_VEL
LIN {X 0,Y 154.196,Z 679.816,A -85,B 0,C 180,E1 -25428.345,E2 -25428.345} C_VEL
LIN {X 0,Y 151.559,Z 692.604,A -85,B 0,C 180,E1 -25429.738,E2 -25429.738} C_VEL
LIN {X 0,Y 148.18,Z 704.418,A -85,B 0,C 180,E1 -25431.502,E2 -25431.502} C_VEL
LIN {X 0,Y 144.437,Z 715.739,A -85,B 0,C 180,E1 -25433.846,E2 -25433.846} C_VEL
LIN {X 0,Y 140.389,Z 725.959,A -85,B 0,C 180,E1 -25436.588,E2 -25436.588} C_VEL
LIN {X 0,Y 136.048,Z 735.152,A -85,B 0,C 180,E1 -25439.758,E2 -25439.758} C_VEL
LIN {X 0,Y 132.24,Z 742.724,A -85,B 0,C 180,E1 -25443.145,E2 -25443.145} C_VEL
LIN {X 0,Y 128.472,Z 750.133,A -85,B 0,C 180,E1 -25447.485,E2 -25447.485} C_VEL
LIN {X 0,Y 125.273,Z 756.09,A -85,B 0,C 180,E1 -25452.028,E2 -25452.028} C_VEL
LIN {X 0,Y 122.74,Z 760.807,A -85,B 0,C 180,E1 -25456.76,E2 -25456.76} C_VEL
LIN {X 0,Y 120.882,Z 764.427,A -85,B 0,C 180,E1 -25461.643,E2 -25461.643} C_VEL
LIN {X 0,Y 119.51,Z 767.836,A -85,B 0,C 180,E1 -25468.668,E2 -25468.668} C_VEL
LIN {X 0,Y 119.286,Z 769.114,A -85,B 0,C 180,E1 -25473.378,E2 -25473.378} C_VEL
LIN {X 0,Y 119.31,Z 769.527,A -85,B 0,C 180,E1 -25476.766,E2 -25476.766} C_VEL
LIN {X 0,Y 119.621,Z 769.56,A -85,B 0,C 180,E1 -25480.152,E2 -25480.152} C_VEL
LIN {X 0,Y 120.223,Z 769.213,A -85,B 0,C 180,E1 -25483.522,E2 -25483.522} C_VEL
LIN {X 0,Y 121.106,Z 768.472,A -85,B 0,C 180,E1 -25486.867,E2 -25486.867} C_VEL
LIN {X 0,Y 122.4,Z 767.288,A -85,B 0,C 180,E1 -25490.151,E2 -25490.151} C_VEL
LIN {X 0,Y 124.974,Z 764.757,A -85,B 0,C 180,E1 -25494.946,E2 -25494.946} C_VEL
LIN {X 0,Y 128.29,Z 761.213,A -85,B 0,C 180,E1 -25499.54,E2 -25499.54} C_VEL
LIN {X 0,Y 132.282,Z 756.55,A -85,B 0,C 180,E1 -25503.906,E2 -25503.906} C_VEL
LIN {X 0,Y 137.041,Z 750.625,A -85,B 0,C 180,E1 -25507.98,E2 -25507.98} C_VEL
LIN {X 0,Y 142.16,Z 743.525,A -85,B 0,C 180,E1 -25511.655,E2 -25511.655} C_VEL
LIN {X 0,Y 147.194,Z 735.665,A -85,B 0,C 180,E1 -25514.768,E2 -25514.768} C_VEL
LIN {X 0,Y 152.408,Z 726.489,A -85,B 0,C 180,E1 -25517.543,E2 -25517.543} C_VEL
LIN {X 0,Y 157.464,Z 716.257,A -85,B 0,C 180,E1 -25519.846,E2 -25519.846} C_VEL
